LIN {X 0,Y 368.794,Z 449.579,A -85,B 0,C 180,E1 -12880.986,E2 -12880.986} C_VEL
LIN {X 0,Y 368.966,Z 448.589,A -85,B 0,C 180,E1 -12882.095,E2 -12882.095} C_VEL
LIN {X 0,Y 369.505,Z 445.744,A -85,B 0,C 180,E1 -12884.062,E2 -12884.062} C_VEL
LIN {X 0,Y 370.092,Z 441.621,A -85,B 0,C 180,E1 -12885.983,E2 -12885.983} C_VEL
LIN {X 0,Y 370.796,Z 436.818,A -85,B 0,C 180,E1 -12887.654,E2 -12887.654} C_VEL
LIN {X 0,Y 371.622,Z 430.934,A -85,B 0,C 180,E1 -12889.269,E2 -12889.269} C_VEL
LIN {X 0,Y 372.743,Z 423.026,A -85,B 0,C 180,E1 -12890.992,E2 -12890.992} C_VEL
LIN {X 0,Y 373.826,Z 414.283,A -85,B 0,C 180,E1 -12892.509,E2 -12892.509} C_VEL
LIN {X 0,Y 374.877,Z 404.263,A -85,B 0,C 180,E1 -12893.917,E2 -12893.917} C_VEL
LIN {X 0,Y 375.773,Z 395.454,A -85,B 0,C 180,E1 -12894.914,E2 -12894.914} C_VEL
LIN {X 0,Y 375.534,Z 390.642,A -85,B 0,C 180,E1 -12895.44,E2 -12895.44} C_VEL
LIN {X 0,Y 373.509,Z 382.744,A -85,B 0,C 180,E1 -12896.307,E2 -12896.307} C_VEL
LIN {X 0,Y 371.458,Z 374.464,A -85,B 0,C 180,E1 -12897.072,E2 -12897.072} C_VEL
LIN {X 0,Y 371.152,Z 369.066,A -85,B 0,C 180,E1 -12897.429,E2 -12897.429} C_VEL
LIN {X 0,Y 371.504,Z 356.306,A -85,B 0,C 180,E1 -12898.033,E2 -12898.033} C_VEL
LIN {X 0,Y 371.686,Z 343.881,A -85,B 0,C 180,E1 -12898.405,E2 -12898.405} C_VEL
LIN {X 0,Y 372.372,Z 304.643,A -85,B 0,C 180,E1 -12899.179,E2 -12899.179} C_VEL
LIN {X 0,Y 372.772,Z 284.426,A -85,B 0,C 180,E1 -12899.575,E2 -12899.575} C_VEL
LIN {X 0,Y 364.309,Z 266.025,A -85,B 0,C 180,E1 -12900.603,E2 -12900.603} C_VEL
LIN {X 0,Y 362.041,Z 261.256,A -85,B 0,C 180,E1 -12900.916,E2 -12900.916} C_VEL
LIN {X 0,Y 361.882,Z 260.447,A -85,B 0,C 180,E1 -12901.182,E2 -12901.182} C_VEL
LIN {X 0,Y 361.852,Z 260.4,A -85,B 0,C 180,E1 -12904.28,E2 -12904.28} C_VEL
LIN {X 0,Y 361.858,Z 260.37,A -85,B 0,C 180,E1 -12907.221,E2 -12907.221} C_VEL
LIN {X 0,Y 361.811,Z 260.413,A -85,B 0,C 180,E1 -12910.75,E2 -12910.75} C_VEL
LIN {X 0,Y 361.811,Z 260.421,A -85,B 0,C 180,E1 -12914.369,E2 -12914.369} C_VEL
LIN {X 0,Y 361.821,Z 260.402,A -85,B 0,C 180,E1 -12917.57,E2 -12917.57} C_VEL
LIN {X 0,Y 361.84,Z 260.396,A -85,B 0,C 180,E1 -12921.571,E2 -12921.571} C_VEL
LIN {X 0,Y 361.872,Z 260.405,A -85,B 0,C 180,E1 -12924.655,E2 -12924.655} C_VEL
LIN {X 0,Y 361.835,Z 260.392,A -85,B 0,C 180,E1 -12928.37,E2 -12928.37} C_VEL
LIN {X 0,Y 361.863,Z 260.391,A -85,B 0,C 180,E1 -12930.952,E2 -12930.952} C_VEL
LIN {X 0,Y 361.872,Z 260.405,A -85,B 0,C 180,E1 -12934.705,E2 -12934.705} C_VEL
LIN {X 0,Y 361.851,Z 260.373,A -85,B 0,C 180,E1 -12938.344,E2 -12938.344} C_VEL
LIN {X 0,Y 361.964,Z 260.396,A -85,B 0,C 180,E1 -12942.061,E2 -12942.061} C_VEL
LIN {X 0,Y 361.994,Z 260.386,A -85,B 0,C 180,E1 -12946.101,E2 -12946.101} C_VEL
LIN {X 0,Y 361.993,Z 260.384,A -85,B 0,C 180,E1 -12949.937,E2 -12949.937} C_VEL
LIN {X 0,Y 362.112,Z 260.378,A -85,B 0,C 180,E1 -12953.312,E2 -12953.312} C_VEL
LIN {X 0,Y 362.257,Z 260.357,A -85,B 0,C 180,E1 -12957.776,E2 -12957.776} C_VEL
LIN {X 0,Y 362.262,Z 260.35,A -85,B 0,C 180,E1 -12962.223,E2 -12962.223} C_VEL
LIN {X 0,Y 362.109,Z 260.371,A -85,B 0,C 180,E1 -12966.687,E2 -12966.687} C_VEL
LIN {X 0,Y 361.993,Z 260.392,A -85,B 0,C 180,E1 -12970.063,E2 -12970.063} C_VEL
LIN {X 0,Y 361.993,Z 260.387,A -85,B 0,C 180,E1 -12973.899,E2 -12973.899} C_VEL
LIN {X 0,Y 361.922,Z 260.403,A -85,B 0,C 180,E1 -12976.934,E2 -12976.934} C_VEL
LIN {X 0,Y 361.878,Z 260.407,A -85,B 0,C 180,E1 -12980.461,E2 -12980.461} C_VEL
LIN {X 0,Y 361.889,Z 260.406,A -85,B 0,C 180,E1 -12984.113,E2 -12984.113} C_VEL
LIN {X 0,Y 361.83,Z 260.393,A -85,B 0,C 180,E1 -12987.785,E2 -12987.785} C_VEL
LIN {X 0,Y 361.822,Z 260.415,A -85,B 0,C 180,E1 -12991.28,E2 -12991.28} C_VEL
LIN {X 0,Y 361.849,Z 260.396,A -85,B 0,C 180,E1 -12994.281,E2 -12994.281} C_VEL
LIN {X 0,Y 361.854,Z 260.408,A -85,B 0,C 180,E1 -12997.222,E2 -12997.222} C_VEL
LIN {X 0,Y 361.807,Z 260.419,A -85,B 0,C 180,E1 -13000.751,E2 -13000.751} C_VEL
LIN {X 0,Y 361.808,Z 260.415,A -85,B 0,C 180,E1 -13004.37,E2 -13004.37} C_VEL
LIN {X 0,Y 361.819,Z 260.416,A -85,B 0,C 180,E1 -13007.571,E2 -13007.571} C_VEL
LIN {X 0,Y 361.839,Z 260.393,A -85,B 0,C 180,E1 -13011.572,E2 -13011.572} C_VEL
LIN {X 0,Y 361.914,Z 260.609,A -85,B 0,C 180,E1 -13015.283,E2 -13015.283} C_VEL
LIN {X 0,Y 364.922,Z 272.495,A -85,B 0,C 180,E1 -13017.929,E2 -13017.929} C_VEL
LIN {X 0,Y 367.637,Z 284.863,A -85,B 0,C 180,E1 -13020.511,E2 -13020.511} C_VEL
LIN {X 0,Y 367.806,Z 288.203,A -85,B 0,C 180,E1 -13021.153,E2 -13021.153} C_VEL
LIN {X 0,Y 365.998,Z 306.761,A -85,B 0,C 180,E1 -13024.49,E2 -13024.49} C_VEL
LIN {X 0,Y 364.837,Z 320.891,A -85,B 0,C 180,E1 -13026.972,E2 -13026.972} C_VEL
LIN {X 0,Y 369.095,Z 349.309,A -85,B 0,C 180,E1 -13027.909,E2 -13027.909} C_VEL
LIN {X 0,Y 371.223,Z 369.3,A -85,B 0,C 180,E1 -13028.472,E2 -13028.472} C_VEL
LIN {X 0,Y 370.056,Z 432.727,A -85,B 0,C 180,E1 -13029.748,E2 -13029.748} C_VEL
LIN {X 0,Y 369.257,Z 446.633,A -85,B 0,C 180,E1 -13030.255,E2 -13030.255} C_VEL
LIN {X 0,Y 368.138,Z 458.947,A -85,B 0,C 180,E1 -13030.918,E2 -13030.918} C_VEL
LIN {X 0,Y 366.661,Z 471.598,A -85,B 0,C 180,E1 -13031.852,E2 -13031.852} C_VEL
LIN {X 0,Y 365.384,Z 482.905,A -85,B 0,C 180,E1 -13032.943,E2 -13032.943} C_VEL
LIN {X 0,Y 364.037,Z 493.136,A -85,B 0,C 180,E1 -13034.175,E2 -13034.175} C_VEL
LIN {X 0,Y 362.945,Z 503.063,A -85,B 0,C 180,E1 -13035.677,E2 -13035.677} C_VEL
LIN {X 0,Y 361.853,Z 512.169,A -85,B 0,C 180,E1 -13037.379,E2 -13037.379} C_VEL
LIN {X 0,Y 361.162,Z 519.379,A -85,B 0,C 180,E1 -13039.063,E2 -13039.063} C_VEL
LIN {X 0,Y 360.78,Z 526.029,A -85,B 0,C 180,E1 -13041.034,E2 -13041.034} C_VEL
LIN {X 0,Y 360.695,Z 530.466,A -85,B 0,C 180,E1 -13042.724,E2 -13042.724} C_VEL
LIN {X 0,Y 360.828,Z 533.844,A -85,B 0,C 180,E1 -13044.411,E2 -13044.411} C_VEL
LIN {X 0,Y 361.054,Z 536.833,A -85,B 0,C 180,E1 -13046.652,E2 -13046.652} C_VEL
LIN {X 0,Y 361.064,Z 537.659,A -85,B 0,C 180,E1 -13047.769,E2 -13047.769} C_VEL
LIN {X 0,Y 361.187,Z 538.105,A -85,B 0,C 180,E1 -13050,E2 -13050} C_VEL
LIN {X 0,Y 361.135,Z 537.717,A -85,B 0,C 180,E1 -13051.115,E2 -13051.115} C_VEL
LIN {X 0,Y 361.114,Z 536.889,A -85,B 0,C 180,E1 -13052.23,E2 -13052.23} C_VEL
LIN {X 0,Y 361.175,Z 535.642,A -85,B 0,C 180,E1 -13053.346,E2 -13053.346} C_VEL
LIN {X 0,Y 360.962,Z 532.923,A -85,B 0,C 180,E1 -13055.026,E2 -13055.026} C_VEL
LIN {X 0,Y 360.858,Z 529.155,A -85,B 0,C 180,E1 -13056.71,E2 -13056.71} C_VEL
LIN {X 0,Y 360.847,Z 524.233,A -85,B 0,C 180,E1 -13058.399,E2 -13058.399} C_VEL
LIN {X 0,Y 361.024,Z 518.022,A -85,B 0,C 180,E1 -13060.09,E2 -13060.09} C_VEL
LIN {X 0,Y 361.441,Z 510.307,A -85,B 0,C 180,E1 -13061.78,E2 -13061.78} C_VEL
LIN {X 0,Y 362.104,Z 502.46,A -85,B 0,C 180,E1 -13063.182,E2 -13063.182} C_VEL
LIN {X 0,Y 362.746,Z 494.101,A -85,B 0,C 180,E1 -13064.422,E2 -13064.422} C_VEL
LIN {X 0,Y 363.596,Z 483.575,A -85,B 0,C 180,E1 -13065.7,E2 -13065.7} C_VEL
LIN {X 0,Y 364.655,Z 472.11,A -85,B 0,C 180,E1 -13066.803,E2 -13066.803} C_VEL
LIN {X 0,Y 365.687,Z 460.234,A -85,B 0,C 180,E1 -13067.691,E2 -13067.691} C_VEL
LIN {X 0,Y 366.606,Z 447.205,A -85,B 0,C 180,E1 -13068.403,E2 -13068.403} C_VEL
LIN {X 0,Y 367.2,Z 433.206,A -85,B 0,C 180,E1 -13068.915,E2 -13068.915} C_VEL
LIN {X 0,Y 368.032,Z 367.575,A -85,B 0,C 180,E1 -13070.214,E2 -13070.214} C_VEL
LIN {X 0,Y 363.351,Z 322.227,A -85,B 0,C 180,E1 -13071.372,E2 -13071.372} C_VEL
LIN {X 0,Y 365.027,Z 297.412,A -85,B 0,C 180,E1 -13075.669,E2 -13075.669} C_VEL
LIN {X 0,Y 366.152,Z 281.581,A -85,B 0,C 180,E1 -13078.452,E2 -13078.452} C_VEL
LIN {X 0,Y 363.857,Z 269.465,A -85,B 0,C 180,E1 -13080.786,E2 -13080.786} C_VEL
LIN {X 0,Y 361.881,Z 260.54,A -85,B 0,C 180,E1 -13082.609,E2 -13082.609} C_VEL
LIN {X 0,Y 361.858,Z 260.411,A -85,B 0,C 180,E1 -13085.636,E2 -13085.636} C_VEL
LIN {X 0,Y 361.818,Z 260.415,A -85,B 0,C 180,E1 -13089.016,E2 -13089.016} C_VEL
LIN {X 0,Y 361.822,Z 260.413,A -85,B 0,C 180,E1 -13092.829,E2 -13092.829} C_VEL
LIN {X 0,Y 361.805,Z 260.414,A -85,B 0,C 180,E1 -13095.947,E2 -13095.947} C_VEL
LIN {X 0,Y 361.802,Z 260.419,A -85,B 0,C 180,E1 -13099.248,E2 -13099.248} C_VEL
LIN {X 0,Y 361.852,Z 260.412,A -85,B 0,C 180,E1 -13102.98,E2 -13102.98} C_VEL
LIN {X 0,Y 361.848,Z 260.41,A -85,B 0,C 180,E1 -13106.631,E2 -13106.631} C_VEL
LIN {X 0,Y 361.837,Z 260.41,A -85,B 0,C 180,E1 -13109.669,E2 -13109.669} C_VEL
LIN {X 0,Y 361.843,Z 260.41,A -85,B 0,C 180,E1 -13113.466,E2 -13113.466} C_VEL
LIN {X 0,Y 361.859,Z 260.407,A -85,B 0,C 180,E1 -13115.93,E2 -13115.93} C_VEL
LIN {X 0,Y 361.865,Z 260.407,A -85,B 0,C 180,E1 -13119.538,E2 -13119.538} C_VEL
LIN {X 0,Y 361.915,Z 260.403,A -85,B 0,C 180,E1 -13123.065,E2 -13123.065} C_VEL
LIN {X 0,Y 361.988,Z 260.395,A -85,B 0,C 180,E1 -13126.528,E2 -13126.528} C_VEL
LIN {X 0,Y 361.985,Z 260.391,A -85,B 0,C 180,E1 -13129.937,E2 -13129.937} C_VEL
LIN {X 0,Y 362.103,Z 260.377,A -85,B 0,C 180,E1 -13133.313,E2 -13133.313} C_VEL
LIN {X 0,Y 362.255,Z 260.358,A -85,B 0,C 180,E1 -13137.777,E2 -13137.777} C_VEL
LIN {X 0,Y 362.244,Z 260.362,A -85,B 0,C 180,E1 -13142.224,E2 -13142.224} C_VEL
LIN {X 0,Y 362.106,Z 260.379,A -85,B 0,C 180,E1 -13146.688,E2 -13146.688} C_VEL
LIN {X 0,Y 361.982,Z 260.395,A -85,B 0,C 180,E1 -13150.064,E2 -13150.064} C_VEL
LIN {X 0,Y 361.988,Z 260.393,A -85,B 0,C 180,E1 -13153.899,E2 -13153.899} C_VEL
LIN {X 0,Y 361.917,Z 260.4,A -85,B 0,C 180,E1 -13156.935,E2 -13156.935} C_VEL
LIN {X 0,Y 361.874,Z 260.408,A -85,B 0,C 180,E1 -13160.462,E2 -13160.462} C_VEL
LIN {X 0,Y 361.852,Z 260.414,A -85,B 0,C 180,E1 -13164.102,E2 -13164.102} C_VEL
LIN {X 0,Y 361.826,Z 260.414,A -85,B 0,C 180,E1 -13167.786,E2 -13167.786} C_VEL
LIN {X 0,Y 361.839,Z 260.41,A -85,B 0,C 180,E1 -13171.286,E2 -13171.286} C_VEL
LIN {X 0,Y 361.843,Z 260.412,A -85,B 0,C 180,E1 -13174.282,E2 -13174.282} C_VEL
LIN {X 0,Y 361.85,Z 260.409,A -85,B 0,C 180,E1 -13177.222,E2 -13177.222} C_VEL
LIN {X 0,Y 361.804,Z 260.414,A -85,B 0,C 180,E1 -13180.752,E2 -13180.752} C_VEL
LIN {X 0,Y 361.805,Z 260.414,A -85,B 0,C 180,E1 -13184.371,E2 -13184.371} C_VEL
LIN {X 0,Y 361.817,Z 260.417,A -85,B 0,C 180,E1 -13187.572,E2 -13187.572} C_VEL
LIN {X 0,Y 361.838,Z 260.415,A -85,B 0,C 180,E1 -13191.573,E2 -13191.573} C_VEL
LIN {X 0,Y 361.867,Z 260.406,A -85,B 0,C 180,E1 -13194.658,E2 -13194.658} C_VEL
LIN {X 0,Y 361.844,Z 260.41,A -85,B 0,C 180,E1 -13197.056,E2 -13197.056} C_VEL
LIN {X 0,Y 361.848,Z 260.409,A -85,B 0,C 180,E1 -13200.952,E2 -13200.952} C_VEL
LIN {X 0,Y 361.859,Z 260.407,A -85,B 0,C 180,E1 -13204.706,E2 -13204.706} C_VEL
LIN {X 0,Y 361.86,Z 260.407,A -85,B 0,C 180,E1 -13208.346,E2 -13208.346} C_VEL
LIN {X 0,Y 361.906,Z 260.401,A -85,B 0,C 180,E1 -13212.094,E2 -13212.094} C_VEL
LIN {X 0,Y 361.953,Z 260.389,A -85,B 0,C 180,E1 -13216.133,E2 -13216.133} C_VEL
LIN {X 0,Y 362.035,Z 260.634,A -85,B 0,C 180,E1 -13216.958,E2 -13216.958} C_VEL
LIN {X 0,Y 362.301,Z 261.741,A -85,B 0,C 180,E1 -13217.125,E2 -13217.125} C_VEL
LIN {X 0,Y 369.26,Z 280.308,A -85,B 0,C 180,E1 -13217.878,E2 -13217.878} C_VEL
LIN {X 0,Y 368.244,Z 347.877,A -85,B 0,C 180,E1 -13219.207,E2 -13219.207} C_VEL
LIN {X 0,Y 368.066,Z 360.994,A -85,B 0,C 180,E1 -13219.689,E2 -13219.689} C_VEL
LIN {X 0,Y 367.703,Z 372.477,A -85,B 0,C 180,E1 -13220.304,E2 -13220.304} C_VEL
LIN {X 0,Y 367.062,Z 384.829,A -85,B 0,C 180,E1 -13221.19,E2 -13221.19} C_VEL
LIN {X 0,Y 366.27,Z 396.386,A -85,B 0,C 180,E1 -13222.282,E2 -13222.282} C_VEL
LIN {X 0,Y 365.484,Z 406.742,A -85,B 0,C 180,E1 -13223.514,E2 -13223.514} C_VEL
LIN {X 0,Y 364.793,Z 415.21,A -85,B 0,C 180,E1 -13224.75,E2 -13224.75} C_VEL
LIN {X 0,Y 364.094,Z 423.021,A -85,B 0,C 180,E1 -13226.127,E2 -13226.127} C_VEL
LIN {X 0,Y 363.274,Z 430.704,A -85,B 0,C 180,E1 -13227.783,E2 -13227.783} C_VEL
LIN {X 0,Y 362.656,Z 436.84,A -85,B 0,C 180,E1 -13229.445,E2 -13229.445} C_VEL
LIN {X 0,Y 362.193,Z 441.726,A -85,B 0,C 180,E1 -13231.112,E2 -13231.112} C_VEL
LIN {X 0,Y 361.837,Z 445.517,A -85,B 0,C 180,E1 -13232.784,E2 -13232.784} C_VEL
LIN {X 0,Y 361.658,Z 448.299,A -85,B 0,C 180,E1 -13234.459,E2 -13234.459} C_VEL
LIN {X 0,Y 361.626,Z 449.614,A -85,B 0,C 180,E1 -13235.577,E2 -13235.577} C_VEL
LIN {X 0,Y 361.569,Z 451.113,A -85,B 0,C 180,E1 -13237.82,E2 -13237.82} C_VEL
LIN {X 0,Y 361.68,Z 450.991,A -85,B 0,C 180,E1 -13240.072,E2 -13240.072} C_VEL
LIN {X 0,Y 361.797,Z 450.359,A -85,B 0,C 180,E1 -13241.201,E2 -13241.201} C_VEL
LIN {X 0,Y 361.982,Z 449.329,A -85,B 0,C 180,E1 -13242.332,E2 -13242.332} C_VEL
LIN {X 0,Y 362.531,Z 446.595,A -85,B 0,C 180,E1 -13244.232,E2 -13244.232} C_VEL
LIN {X 0,Y 363.212,Z 442.213,A -85,B 0,C 180,E1 -13246.294,E2 -13246.294} C_VEL
LIN {X 0,Y 363.955,Z 437.339,A -85,B 0,C 180,E1 -13247.997,E2 -13247.997} C_VEL
LIN {X 0,Y 364.868,Z 431.376,A -85,B 0,C 180,E1 -13249.641,E2 -13249.641} C_VEL
LIN {X 0,Y 365.853,Z 424.772,A -85,B 0,C 180,E1 -13251.112,E2 -13251.112} C_VEL
LIN {X 0,Y 367.027,Z 415.918,A -85,B 0,C 180,E1 -13252.709,E2 -13252.709} C_VEL
LIN {X 0,Y 368.04,Z 406.472,A -85,B 0,C 180,E1 -13254.09,E2 -13254.09} C_VEL
LIN {X 0,Y 369.221,Z 395.597,A -85,B 0,C 180,E1 -13255.358,E2 -13255.358} C_VEL
LIN {X 0,Y 370.101,Z 385.806,A -85,B 0,C 180,E1 -13256.27,E2 -13256.27} C_VEL
LIN {X 0,Y 370.899,Z 374.104,A -85,B 0,C 180,E1 -13257.126,E2 -13257.126} C_VEL
LIN {X 0,Y 371.152,Z 369.066,A -85,B 0,C 180,E1 -13257.429,E2 -13257.429} C_VEL
LIN {X 0,Y 370.716,Z 365.396,A -85,B 0,C 180,E1 -13257.67,E2 -13257.67} C_VEL
LIN {X 0,Y 365.698,Z 354.113,A -85,B 0,C 180,E1 -13258.532,E2 -13258.532} C_VEL
LIN {X 0,Y 365.154,Z 350.323,A -85,B 0,C 180,E1 -13258.697,E2 -13258.697} C_VEL
LIN {X 0,Y 365.736,Z 311.849,A -85,B 0,C 180,E1 -13259.507,E2 -13259.507} C_VEL
LIN {X 0,Y 366.277,Z 286.132,A -85,B 0,C 180,E1 -13260.019,E2 -13260.019} C_VEL
LIN {X 0,Y 357.814,Z 267.909,A -85,B 0,C 180,E1 -13261.076,E2 -13261.076} C_VEL
LIN {X 0,Y 355.007,Z 262.187,A -85,B 0,C 180,E1 -13261.458,E2 -13261.458} C_VEL
LIN {X 0,Y 354.799,Z 261.368,A -85,B 0,C 180,E1 -13261.702,E2 -13261.702} C_VEL
LIN {X 0,Y 354.809,Z 261.256,A -85,B 0,C 180,E1 -13265.059,E2 -13265.059} C_VEL
LIN {X 0,Y 354.793,Z 261.258,A -85,B 0,C 180,E1 -13267.884,E2 -13267.884} C_VEL
LIN {X 0,Y 354.769,Z 261.286,A -85,B 0,C 180,E1 -13271.167,E2 -13271.167} C_VEL
LIN {X 0,Y 354.758,Z 261.299,A -85,B 0,C 180,E1 -13274.505,E2 -13274.505} C_VEL
LIN {X 0,Y 354.78,Z 261.279,A -85,B 0,C 180,E1 -13277.66,E2 -13277.66} C_VEL
LIN {X 0,Y 354.784,Z 261.284,A -85,B 0,C 180,E1 -13280.661,E2 -13280.661} C_VEL
LIN {X 0,Y 354.819,Z 261.278,A -85,B 0,C 180,E1 -13284.3,E2 -13284.3} C_VEL
LIN {X 0,Y 354.785,Z 261.281,A -85,B 0,C 180,E1 -13287.666,E2 -13287.666} C_VEL
LIN {X 0,Y 354.796,Z 261.279,A -85,B 0,C 180,E1 -13291.614,E2 -13291.614} C_VEL
LIN {X 0,Y 354.837,Z 261.279,A -85,B 0,C 180,E1 -13295.422,E2 -13295.422} C_VEL
LIN {X 0,Y 354.821,Z 261.253,A -85,B 0,C 180,E1 -13299.112,E2 -13299.112} C_VEL
LIN {X 0,Y 354.895,Z 261.277,A -85,B 0,C 180,E1 -13302.719,E2 -13302.719} C_VEL
LIN {X 0,Y 354.947,Z 261.265,A -85,B 0,C 180,E1 -13306.255,E2 -13306.255} C_VEL
LIN {X 0,Y 354.95,Z 261.263,A -85,B 0,C 180,E1 -13309.735,E2 -13309.735} C_VEL
LIN {X 0,Y 355.079,Z 261.253,A -85,B 0,C 180,E1 -13313.179,E2 -13313.179} C_VEL
LIN {X 0,Y 355.219,Z 261.233,A -85,B 0,C 180,E1 -13317.732,E2 -13317.732} C_VEL
LIN {X 0,Y 355.139,Z 261.239,A -85,B 0,C 180,E1 -13321.134,E2 -13321.134} C_VEL
LIN {X 0,Y 355.224,Z 261.226,A -85,B 0,C 180,E1 -13322.268,E2 -13322.268} C_VEL
LIN {X 0,Y 355.076,Z 261.247,A -85,B 0,C 180,E1 -13326.82,E2 -13326.82} C_VEL
LIN {X 0,Y 354.949,Z 261.269,A -85,B 0,C 180,E1 -13330.265,E2 -13330.265} C_VEL
LIN {X 0,Y 354.938,Z 261.267,A -85,B 0,C 180,E1 -13334.018,E2 -13334.018} C_VEL
LIN {X 0,Y 354.885,Z 261.272,A -85,B 0,C 180,E1 -13338.092,E2 -13338.092} C_VEL
LIN {X 0,Y 354.812,Z 261.284,A -85,B 0,C 180,E1 -13341.417,E2 -13341.417} C_VEL
LIN {X 0,Y 354.843,Z 261.284,A -85,B 0,C 180,E1 -13344.577,E2 -13344.577} C_VEL
LIN {X 0,Y 354.784,Z 261.274,A -85,B 0,C 180,E1 -13348.387,E2 -13348.387} C_VEL
LIN {X 0,Y 354.775,Z 261.288,A -85,B 0,C 180,E1 -13352.335,E2 -13352.335} C_VEL
LIN {X 0,Y 354.817,Z 261.287,A -85,B 0,C 180,E1 -13355.699,E2 -13355.699} C_VEL
LIN {X 0,Y 354.765,Z 261.285,A -85,B 0,C 180,E1 -13359.413,E2 -13359.413} C_VEL
LIN {X 0,Y 354.778,Z 261.285,A -85,B 0,C 180,E1 -13362.866,E2 -13362.866} C_VEL
LIN {X 0,Y 354.759,Z 261.29,A -85,B 0,C 180,E1 -13366.103,E2 -13366.103} C_VEL
LIN {X 0,Y 354.76,Z 261.286,A -85,B 0,C 180,E1 -13369.176,E2 -13369.176} C_VEL
LIN {X 0,Y 354.796,Z 261.284,A -85,B 0,C 180,E1 -13372.405,E2 -13372.405} C_VEL
LIN {X 0,Y 354.867,Z 261.516,A -85,B 0,C 180,E1 -13374.808,E2 -13374.808} C_VEL
LIN {X 0,Y 357.964,Z 273.72,A -85,B 0,C 180,E1 -13377.59,E2 -13377.59} C_VEL
LIN {X 0,Y 360.672,Z 285.936,A -85,B 0,C 180,E1 -13380.206,E2 -13380.206} C_VEL
LIN {X 0,Y 361.002,Z 289.292,A -85,B 0,C 180,E1 -13380.876,E2 -13380.876} C_VEL
LIN {X 0,Y 359.358,Z 305.33,A -85,B 0,C 180,E1 -13383.817,E2 -13383.817} C_VEL
LIN {X 0,Y 358.071,Z 319.999,A -85,B 0,C 180,E1 -13386.444,E2 -13386.444} C_VEL
LIN {X 0,Y 362.388,Z 348.333,A -85,B 0,C 180,E1 -13387.415,E2 -13387.415} C_VEL
LIN {X 0,Y 364.682,Z 369.563,A -85,B 0,C 180,E1 -13388.031,E2 -13388.031} C_VEL
LIN {X 0,Y 363.49,Z 431.442,A -85,B 0,C 180,E1 -13389.293,E2 -13389.293} C_VEL
LIN {X 0,Y 362.782,Z 444.691,A -85,B 0,C 180,E1 -13389.777,E2 -13389.777} C_VEL
LIN {X 0,Y 361.649,Z 456.751,A -85,B 0,C 180,E1 -13390.414,E2 -13390.414} C_VEL
LIN {X 0,Y 360.359,Z 468.169,A -85,B 0,C 180,E1 -13391.228,E2 -13391.228} C_VEL
LIN {X 0,Y 358.911,Z 479.95,A -85,B 0,C 180,E1 -13392.331,E2 -13392.331} C_VEL
LIN {X 0,Y 357.475,Z 490.561,A -85,B 0,C 180,E1 -13393.584,E2 -13393.584} C_VEL
LIN {X 0,Y 356.349,Z 499.279,A -85,B 0,C 180,E1 -13394.852,E2 -13394.852} C_VEL
LIN {X 0,Y 355.493,Z 507.367,A -85,B 0,C 180,E1 -13396.276,E2 -13396.276} C_VEL
LIN {X 0,Y 354.644,Z 514.098,A -85,B 0,C 180,E1 -13397.7,E2 -13397.7} C_VEL
LIN {X 0,Y 353.935,Z 520.776,A -85,B 0,C 180,E1 -13399.416,E2 -13399.416} C_VEL
LIN {X 0,Y 353.667,Z 526.917,A -85,B 0,C 180,E1 -13401.429,E2 -13401.429} C_VEL
LIN {X 0,Y 353.709,Z 531.549,A -85,B 0,C 180,E1 -13403.451,E2 -13403.451} C_VEL
LIN {X 0,Y 353.808,Z 534.75,A -85,B 0,C 180,E1 -13405.442,E2 -13405.442} C_VEL
LIN {X 0,Y 353.977,Z 536.023,A -85,B 0,C 180,E1 -13406.585,E2 -13406.585} C_VEL
LIN {X 0,Y 354.014,Z 536.829,A -85,B 0,C 180,E1 -13407.724,E2 -13407.724} C_VEL
LIN {X 0,Y 354.138,Z 537.248,A -85,B 0,C 180,E1 -13410,E2 -13410} C_VEL
LIN {X 0,Y 354.084,Z 536.842,A -85,B 0,C 180,E1 -13411.137,E2 -13411.137} C_VEL
LIN {X 0,Y 354.064,Z 535.988,A -85,B 0,C 180,E1 -13412.275,E2 -13412.275} C_VEL
LIN {X 0,Y 354.129,Z 534.725,A -85,B 0,C 180,E1 -13413.413,E2 -13413.413} C_VEL
LIN {X 0,Y 353.882,Z 531.968,A -85,B 0,C 180,E1 -13415.127,E2 -13415.127} C_VEL
LIN {X 0,Y 353.771,Z 528.163,A -85,B 0,C 180,E1 -13416.845,E2 -13416.845} C_VEL
LIN {X 0,Y 353.776,Z 523.202,A -85,B 0,C 180,E1 -13418.568,E2 -13418.568} C_VEL
LIN {X 0,Y 353.963,Z 516.946,A -85,B 0,C 180,E1 -13420.293,E2 -13420.293} C_VEL
LIN {X 0,Y 354.412,Z 509.183,A -85,B 0,C 180,E1 -13422.017,E2 -13422.017} C_VEL
LIN {X 0,Y 355.112,Z 501.278,A -85,B 0,C 180,E1 -13423.446,E2 -13423.446} C_VEL
LIN {X 0,Y 355.76,Z 493.258,A -85,B 0,C 180,E1 -13424.654,E2 -13424.654} C_VEL
LIN {X 0,Y 356.593,Z 483.526,A -85,B 0,C 180,E1 -13425.869,E2 -13425.869} C_VEL
LIN {X 0,Y 357.66,Z 472.237,A -85,B 0,C 180,E1 -13426.994,E2 -13426.994} C_VEL
LIN {X 0,Y 358.829,Z 459.612,A -85,B 0,C 180,E1 -13427.967,E2 -13427.967} C_VEL
LIN {X 0,Y 359.731,Z 446.686,A -85,B 0,C 180,E1 -13428.694,E2 -13428.694} C_VEL
LIN {X 0,Y 360.329,Z 434.005,A -85,B 0,C 180,E1 -13429.178,E2 -13429.178} C_VEL
LIN {X 0,Y 360.743,Z 410.493,A -85,B 0,C 180,E1 -13429.688,E2 -13429.688} C_VEL
LIN {X 0,Y 361.236,Z 368.258,A -85,B 0,C 180,E1 -13430.523,E2 -13430.523} C_VEL
LIN {X 0,Y 356.406,Z 321.507,A -85,B 0,C 180,E1 -13431.736,E2 -13431.736} C_VEL
LIN {X 0,Y 357.944,Z 299.576,A -85,B 0,C 180,E1 -13435.591,E2 -13435.591} C_VEL
LIN {X 0,Y 359.183,Z 283.797,A -85,B 0,C 180,E1 -13438.413,E2 -13438.413} C_VEL
LIN {X 0,Y 358.559,Z 278.956,A -85,B 0,C 180,E1 -13439.34,E2 -13439.34} C_VEL
LIN {X 0,Y 355.509,Z 264.371,A -85,B 0,C 180,E1 -13442.258,E2 -13442.258} C_VEL
LIN {X 0,Y 354.823,Z 261.415,A -85,B 0,C 180,E1 -13442.918,E2 -13442.918} C_VEL
LIN {X 0,Y 354.786,Z 261.288,A -85,B 0,C 180,E1 -13446.459,E2 -13446.459} C_VEL
LIN {X 0,Y 354.763,Z 261.296,A -85,B 0,C 180,E1 -13449.411,E2 -13449.411} C_VEL
LIN {X 0,Y 354.774,Z 261.292,A -85,B 0,C 180,E1 -13452.865,E2 -13452.865} C_VEL
LIN {X 0,Y 354.754,Z 261.291,A -85,B 0,C 180,E1 -13456.102,E2 -13456.102} C_VEL
LIN {X 0,Y 354.755,Z 261.298,A -85,B 0,C 180,E1 -13459.175,E2 -13459.175} C_VEL
LIN {X 0,Y 354.79,Z 261.287,A -85,B 0,C 180,E1 -13462.404,E2 -13462.404} C_VEL
LIN {X 0,Y 354.799,Z 261.291,A -85,B 0,C 180,E1 -13464.939,E2 -13464.939} C_VEL
LIN {X 0,Y 354.766,Z 261.29,A -85,B 0,C 180,E1 -13468.409,E2 -13468.409} C_VEL
LIN {X 0,Y 354.778,Z 261.29,A -85,B 0,C 180,E1 -13471.613,E2 -13471.613} C_VEL
LIN {X 0,Y 354.824,Z 261.283,A -85,B 0,C 180,E1 -13475.657,E2 -13475.657} C_VEL
LIN {X 0,Y 354.811,Z 261.288,A -85,B 0,C 180,E1 -13479.112,E2 -13479.112} C_VEL
LIN {X 0,Y 354.868,Z 261.282,A -85,B 0,C 180,E1 -13482.719,E2 -13482.719} C_VEL
LIN {X 0,Y 354.94,Z 261.27,A -85,B 0,C 180,E1 -13486.255,E2 -13486.255} C_VEL
LIN {X 0,Y 354.941,Z 261.268,A -85,B 0,C 180,E1 -13489.735,E2 -13489.735} C_VEL
LIN {X 0,Y 355.07,Z 261.254,A -85,B 0,C 180,E1 -13493.18,E2 -13493.18} C_VEL
LIN {X 0,Y 355.217,Z 261.234,A -85,B 0,C 180,E1 -13497.732,E2 -13497.732} C_VEL
LIN {X 0,Y 355.158,Z 261.242,A -85,B 0,C 180,E1 -13501.134,E2 -13501.134} C_VEL
LIN {X 0,Y 355.206,Z 261.239,A -85,B 0,C 180,E1 -13502.268,E2 -13502.268} C_VEL
LIN {X 0,Y 355.072,Z 261.254,A -85,B 0,C 180,E1 -13506.821,E2 -13506.821} C_VEL
LIN {X 0,Y 354.939,Z 261.274,A -85,B 0,C 180,E1 -13510.266,E2 -13510.266} C_VEL
LIN {X 0,Y 354.932,Z 261.273,A -85,B 0,C 180,E1 -13514.019,E2 -13514.019} C_VEL
LIN {X 0,Y 354.881,Z 261.28,A -85,B 0,C 180,E1 -13518.093,E2 -13518.093} C_VEL
LIN {X 0,Y 354.804,Z 261.292,A -85,B 0,C 180,E1 -13522.108,E2 -13522.108} C_VEL
LIN {X 0,Y 354.793,Z 261.29,A -85,B 0,C 180,E1 -13525.836,E2 -13525.836} C_VEL
LIN {X 0,Y 354.785,Z 261.291,A -85,B 0,C 180,E1 -13529.685,E2 -13529.685} C_VEL
LIN {X 0,Y 354.779,Z 261.291,A -85,B 0,C 180,E1 -13532.335,E2 -13532.335} C_VEL
LIN {X 0,Y 354.811,Z 261.288,A -85,B 0,C 180,E1 -13535.699,E2 -13535.699} C_VEL
LIN {X 0,Y 354.762,Z 261.293,A -85,B 0,C 180,E1 -13539.414,E2 -13539.414} C_VEL
LIN {X 0,Y 354.775,Z 261.287,A -85,B 0,C 180,E1 -13542.867,E2 -13542.867} C_VEL
LIN {X 0,Y 354.757,Z 261.294,A -85,B 0,C 180,E1 -13546.104,E2 -13546.104} C_VEL
LIN {X 0,Y 354.758,Z 261.293,A -85,B 0,C 180,E1 -13549.177,E2 -13549.177} C_VEL
LIN {X 0,Y 354.795,Z 261.285,A -85,B 0,C 180,E1 -13552.406,E2 -13552.406} C_VEL
LIN {X 0,Y 354.805,Z 261.286,A -85,B 0,C 180,E1 -13554.942,E2 -13554.942} C_VEL
LIN {X 0,Y 354.774,Z 261.289,A -85,B 0,C 180,E1 -13558.411,E2 -13558.411} C_VEL
LIN {X 0,Y 354.787,Z 261.293,A -85,B 0,C 180,E1 -13561.615,E2 -13561.615} C_VEL
LIN {X 0,Y 354.804,Z 261.291,A -85,B 0,C 180,E1 -13565.421,E2 -13565.421} C_VEL
LIN {X 0,Y 354.82,Z 261.287,A -85,B 0,C 180,E1 -13569.114,E2 -13569.114} C_VEL
LIN {X 0,Y 354.852,Z 261.281,A -85,B 0,C 180,E1 -13572.718,E2 -13572.718} C_VEL
LIN {X 0,Y 354.967,Z 261.43,A -85,B 0,C 180,E1 -13576.548,E2 -13576.548} C_VEL
LIN {X 0,Y 355.229,Z 262.533,A -85,B 0,C 180,E1 -13576.748,E2 -13576.748} C_VEL
LIN {X 0,Y 362.316,Z 281.131,A -85,B 0,C 180,E1 -13577.535,E2 -13577.535} C_VEL
LIN {X 0,Y 361.46,Z 348.669,A -85,B 0,C 180,E1 -13578.896,E2 -13578.896} C_VEL
LIN {X 0,Y 361.28,Z 361.801,A -85,B 0,C 180,E1 -13579.386,E2 -13579.386} C_VEL
LIN {X 0,Y 360.919,Z 372.74,A -85,B 0,C 180,E1 -13579.978,E2 -13579.978} C_VEL
LIN {X 0,Y 360.269,Z 385.221,A -85,B 0,C 180,E1 -13580.881,E2 -13580.881} C_VEL
LIN {X 0,Y 359.439,Z 396.896,A -85,B 0,C 180,E1 -13581.993,E2 -13581.993} C_VEL
LIN {X 0,Y 358.611,Z 407.313,A -85,B 0,C 180,E1 -13583.248,E2 -13583.248} C_VEL
LIN {X 0,Y 357.825,Z 416.699,A -85,B 0,C 180,E1 -13584.647,E2 -13584.647} C_VEL
LIN {X 0,Y 357.096,Z 424.404,A -85,B 0,C 180,E1 -13586.051,E2 -13586.051} C_VEL
LIN {X 0,Y 356.249,Z 431.955,A -85,B 0,C 180,E1 -13587.739,E2 -13587.739} C_VEL
LIN {X 0,Y 355.625,Z 438.014,A -85,B 0,C 180,E1 -13589.434,E2 -13589.434} C_VEL
LIN {X 0,Y 355.154,Z 442.831,A -85,B 0,C 180,E1 -13591.134,E2 -13591.134} C_VEL
LIN {X 0,Y 354.791,Z 446.558,A -85,B 0,C 180,E1 -13592.839,E2 -13592.839} C_VEL
LIN {X 0,Y 354.616,Z 449.279,A -85,B 0,C 180,E1 -13594.547,E2 -13594.547} C_VEL
LIN {X 0,Y 354.576,Z 450.567,A -85,B 0,C 180,E1 -13595.688,E2 -13595.688} C_VEL
LIN {X 0,Y 354.537,Z 451.859,A -85,B 0,C 180,E1 -13597.623,E2 -13597.623} C_VEL
LIN {X 0,Y 354.565,Z 452.083,A -85,B 0,C 180,E1 -13599.124,E2 -13599.124} C_VEL
LIN {X 0,Y 354.811,Z 451.139,A -85,B 0,C 180,E1 -13601.425,E2 -13601.425} C_VEL
LIN {X 0,Y 355.003,Z 450.053,A -85,B 0,C 180,E1 -13602.578,E2 -13602.578} C_VEL
LIN {X 0,Y 355.572,Z 447.433,A -85,B 0,C 180,E1 -13604.416,E2 -13604.416} C_VEL
LIN {X 0,Y 356.331,Z 442.808,A -85,B 0,C 180,E1 -13606.618,E2 -13606.618} C_VEL
LIN {X 0,Y 357.131,Z 437.863,A -85,B 0,C 180,E1 -13608.353,E2 -13608.353} C_VEL
LIN {X 0,Y 358.156,Z 431.579,A -85,B 0,C 180,E1 -13610.084,E2 -13610.084} C_VEL
LIN {X 0,Y 359.347,Z 423.639,A -85,B 0,C 180,E1 -13611.814,E2 -13611.814} C_VEL
LIN {X 0,Y 360.484,Z 415.52,A -85,B 0,C 180,E1 -13613.247,E2 -13613.247} C_VEL
LIN {X 0,Y 361.619,Z 405.455,A -85,B 0,C 180,E1 -13614.699,E2 -13614.699} C_VEL
LIN {X 0,Y 362.696,Z 395.415,A -85,B 0,C 180,E1 -13615.848,E2 -13615.848} C_VEL
LIN {X 0,Y 363.713,Z 384.542,A -85,B 0,C 180,E1 -13616.839,E2 -13616.839} C_VEL
LIN {X 0,Y 364.415,Z 374.426,A -85,B 0,C 180,E1 -13617.571,E2 -13617.571} C_VEL
LIN {X 0,Y 364.932,Z 361.686,A -85,B 0,C 180,E1 -13618.27,E2 -13618.27} C_VEL
LIN {X 0,Y 365.154,Z 350.323,A -85,B 0,C 180,E1 -13618.697,E2 -13618.697} C_VEL
LIN {X 0,Y 364.696,Z 344.57,A -85,B 0,C 180,E1 -13618.899,E2 -13618.899} C_VEL
LIN {X 0,Y 359.585,Z 326.01,A -85,B 0,C 180,E1 -13619.668,E2 -13619.668} C_VEL
LIN {X 0,Y 359.093,Z 320.207,A -85,B 0,C 180,E1 -13619.824,E2 -13619.824} C_VEL
LIN {X 0,Y 359.844,Z 288.07,A -85,B 0,C 180,E1 -13620.47,E2 -13620.47} C_VEL
LIN {X 0,Y 351.908,Z 271.09,A -85,B 0,C 180,E1 -13621.49,E2 -13621.49} C_VEL
LIN {X 0,Y 347.975,Z 263.262,A -85,B 0,C 180,E1 -13622.02,E2 -13622.02} C_VEL
LIN {X 0,Y 347.789,Z 262.295,A -85,B 0,C 180,E1 -13622.239,E2 -13622.239} C_VEL
LIN {X 0,Y 347.767,Z 262.12,A -85,B 0,C 180,E1 -13626.063,E2 -13626.063} C_VEL
LIN {X 0,Y 347.731,Z 262.158,A -85,B 0,C 180,E1 -13628.795,E2 -13628.795} C_VEL
LIN {X 0,Y 347.742,Z 262.156,A -85,B 0,C 180,E1 -13631.831,E2 -13631.831} C_VEL
LIN {X 0,Y 347.7,Z 262.173,A -85,B 0,C 180,E1 -13635.027,E2 -13635.027} C_VEL
LIN {X 0,Y 347.737,Z 262.163,A -85,B 0,C 180,E1 -13638.399,E2 -13638.399} C_VEL
LIN {X 0,Y 347.76,Z 262.144,A -85,B 0,C 180,E1 -13642.013,E2 -13642.013} C_VEL
LIN {X 0,Y 347.743,Z 262.169,A -85,B 0,C 180,E1 -13645.535,E2 -13645.535} C_VEL
LIN {X 0,Y 347.742,Z 262.147,A -85,B 0,C 180,E1 -13648.3,E2 -13648.3} C_VEL
LIN {X 0,Y 347.742,Z 262.148,A -85,B 0,C 180,E1 -13650.984,E2 -13650.984} C_VEL
LIN {X 0,Y 347.743,Z 262.17,A -85,B 0,C 180,E1 -13653.6,E2 -13653.6} C_VEL
LIN {X 0,Y 347.753,Z 262.147,A -85,B 0,C 180,E1 -13656.159,E2 -13656.159} C_VEL
LIN {X 0,Y 347.801,Z 262.136,A -85,B 0,C 180,E1 -13659.908,E2 -13659.908} C_VEL
LIN {X 0,Y 347.863,Z 262.155,A -85,B 0,C 180,E1 -13662.359,E2 -13662.359} C_VEL
LIN {X 0,Y 347.894,Z 262.141,A -85,B 0,C 180,E1 -13665.97,E2 -13665.97} C_VEL
LIN {X 0,Y 347.89,Z 262.145,A -85,B 0,C 180,E1 -13669.524,E2 -13669.524} C_VEL
LIN {X 0,Y 348.046,Z 262.128,A -85,B 0,C 180,E1 -13673.041,E2 -13673.041} C_VEL
LIN {X 0,Y 348.18,Z 262.109,A -85,B 0,C 180,E1 -13677.686,E2 -13677.686} C_VEL
LIN {X 0,Y 348.11,Z 262.114,A -85,B 0,C 180,E1 -13681.157,E2 -13681.157} C_VEL
LIN {X 0,Y 348.186,Z 262.103,A -85,B 0,C 180,E1 -13682.313,E2 -13682.313} C_VEL
LIN {X 0,Y 348.043,Z 262.121,A -85,B 0,C 180,E1 -13686.959,E2 -13686.959} C_VEL
LIN {X 0,Y 347.889,Z 262.148,A -85,B 0,C 180,E1 -13690.475,E2 -13690.475} C_VEL
LIN {X 0,Y 347.894,Z 262.145,A -85,B 0,C 180,E1 -13694.15,E2 -13694.15} C_VEL
LIN {X 0,Y 347.825,Z 262.151,A -85,B 0,C 180,E1 -13698.259,E2 -13698.259} C_VEL
LIN {X 0,Y 347.758,Z 262.161,A -85,B 0,C 180,E1 -13701.624,E2 -13701.624} C_VEL
LIN {X 0,Y 347.761,Z 262.164,A -85,B 0,C 180,E1 -13705.112,E2 -13705.112} C_VEL
LIN {X 0,Y 347.736,Z 262.157,A -85,B 0,C 180,E1 -13709.016,E2 -13709.016} C_VEL
LIN {X 0,Y 347.726,Z 262.155,A -85,B 0,C 180,E1 -13713.073,E2 -13713.073} C_VEL
LIN {X 0,Y 347.764,Z 262.165,A -85,B 0,C 180,E1 -13716.065,E2 -13716.065} C_VEL
LIN {X 0,Y 347.727,Z 262.159,A -85,B 0,C 180,E1 -13718.796,E2 -13718.796} C_VEL
LIN {X 0,Y 347.736,Z 262.169,A -85,B 0,C 180,E1 -13721.832,E2 -13721.832} C_VEL
LIN {X 0,Y 347.698,Z 262.176,A -85,B 0,C 180,E1 -13725.028,E2 -13725.028} C_VEL
LIN {X 0,Y 347.735,Z 262.171,A -85,B 0,C 180,E1 -13728.4,E2 -13728.4} C_VEL
LIN {X 0,Y 347.759,Z 262.151,A -85,B 0,C 180,E1 -13732.014,E2 -13732.014} C_VEL
LIN {X 0,Y 347.81,Z 262.356,A -85,B 0,C 180,E1 -13734.284,E2 -13734.284} C_VEL
LIN {X 0,Y 351.08,Z 275.148,A -85,B 0,C 180,E1 -13737.283,E2 -13737.283} C_VEL
LIN {X 0,Y 353.702,Z 287.071,A -85,B 0,C 180,E1 -13739.895,E2 -13739.895} C_VEL
LIN {X 0,Y 354.159,Z 290.933,A -85,B 0,C 180,E1 -13740.692,E2 -13740.692} C_VEL
LIN {X 0,Y 352.448,Z 306.991,A -85,B 0,C 180,E1 -13743.694,E2 -13743.694} C_VEL
LIN {X 0,Y 351.311,Z 319.1,A -85,B 0,C 180,E1 -13745.893,E2 -13745.893} C_VEL
LIN {X 0,Y 353.802,Z 334.826,A -85,B 0,C 180,E1 -13746.48,E2 -13746.48} C_VEL
LIN {X 0,Y 357.079,Z 358.789,A -85,B 0,C 180,E1 -13747.254,E2 -13747.254} C_VEL
LIN {X 0,Y 358.272,Z 372.133,A -85,B 0,C 180,E1 -13747.632,E2 -13747.632} C_VEL
LIN {X 0,Y 356.997,Z 430.117,A -85,B 0,C 180,E1 -13748.822,E2 -13748.822} C_VEL
LIN {X 0,Y 356.27,Z 443.53,A -85,B 0,C 180,E1 -13749.315,E2 -13749.315} C_VEL
LIN {X 0,Y 354.971,Z 456.787,A -85,B 0,C 180,E1 -13750.03,E2 -13750.03} C_VEL
LIN {X 0,Y 353.652,Z 467.958,A -85,B 0,C 180,E1 -13750.859,E2 -13750.859} C_VEL
LIN {X 0,Y 352.308,Z 478.305,A -85,B 0,C 180,E1 -13751.839,E2 -13751.839} C_VEL
LIN {X 0,Y 350.808,Z 489.046,A -85,B 0,C 180,E1 -13753.113,E2 -13753.113} C_VEL
LIN {X 0,Y 349.448,Z 498.766,A -85,B 0,C 180,E1 -13754.545,E2 -13754.545} C_VEL
LIN {X 0,Y 348.533,Z 506.793,A -85,B 0,C 180,E1 -13755.997,E2 -13755.997} C_VEL
LIN {X 0,Y 347.64,Z 513.472,A -85,B 0,C 180,E1 -13757.448,E2 -13757.448} C_VEL
LIN {X 0,Y 347.027,Z 519.075,A -85,B 0,C 180,E1 -13758.907,E2 -13758.907} C_VEL
LIN {X 0,Y 346.647,Z 524.61,A -85,B 0,C 180,E1 -13760.665,E2 -13760.665} C_VEL
LIN {X 0,Y 346.531,Z 528.978,A -85,B 0,C 180,E1 -13762.425,E2 -13762.425} C_VEL
LIN {X 0,Y 346.674,Z 532.296,A -85,B 0,C 180,E1 -13764.182,E2 -13764.182} C_VEL
LIN {X 0,Y 346.725,Z 533.961,A -85,B 0,C 180,E1 -13765.349,E2 -13765.349} C_VEL
LIN {X 0,Y 346.901,Z 535.209,A -85,B 0,C 180,E1 -13766.515,E2 -13766.515} C_VEL
LIN {X 0,Y 346.964,Z 536.001,A -85,B 0,C 180,E1 -13767.678,E2 -13767.678} C_VEL
LIN {X 0,Y 347.088,Z 536.391,A -85,B 0,C 180,E1 -13770,E2 -13770} C_VEL
LIN {X 0,Y 347.033,Z 535.961,A -85,B 0,C 180,E1 -13771.16,E2 -13771.16} C_VEL
LIN {X 0,Y 347.016,Z 535.085,A -85,B 0,C 180,E1 -13772.321,E2 -13772.321} C_VEL
LIN {X 0,Y 347.064,Z 533.804,A -85,B 0,C 180,E1 -13773.482,E2 -13773.482} C_VEL
LIN {X 0,Y 346.805,Z 531.012,A -85,B 0,C 180,E1 -13775.232,E2 -13775.232} C_VEL
LIN {X 0,Y 346.692,Z 527.168,A -85,B 0,C 180,E1 -13776.986,E2 -13776.986} C_VEL
LIN {X 0,Y 346.695,Z 522.166,A -85,B 0,C 180,E1 -13778.744,E2 -13778.744} C_VEL
LIN {X 0,Y 346.898,Z 515.866,A -85,B 0,C 180,E1 -13780.505,E2 -13780.505} C_VEL
LIN {X 0,Y 347.395,Z 508.05,A -85,B 0,C 180,E1 -13782.263,E2 -13782.263} C_VEL
LIN {X 0,Y 348.099,Z 500.07,A -85,B 0,C 180,E1 -13783.722,E2 -13783.722} C_VEL
LIN {X 0,Y 348.871,Z 491.433,A -85,B 0,C 180,E1 -13785.029,E2 -13785.029} C_VEL
LIN {X 0,Y 349.891,Z 480.858,A -85,B 0,C 180,E1 -13786.331,E2 -13786.331} C_VEL
LIN {X 0,Y 350.998,Z 469.156,A -85,B 0,C 180,E1 -13787.477,E2 -13787.477} C_VEL
LIN {X 0,Y 352.145,Z 456.835,A -85,B 0,C 180,E1 -13788.395,E2 -13788.395} C_VEL
LIN {X 0,Y 353.062,Z 443.082,A -85,B 0,C 180,E1 -13789.136,E2 -13789.136} C_VEL
LIN {X 0,Y 353.632,Z 430.058,A -85,B 0,C 180,E1 -13789.594,E2 -13789.594} C_VEL
LIN {X 0,Y 354.51,Z 369.681,A -85,B 0,C 180,E1 -13790.825,E2 -13790.825} C_VEL
LIN {X 0,Y 349.518,Z 320.346,A -85,B 0,C 180,E1 -13792.148,E2 -13792.148} C_VEL
LIN {X 0,Y 351.29,Z 296.652,A -85,B 0,C 180,E1 -13796.431,E2 -13796.431} C_VEL
LIN {X 0,Y 352.239,Z 284.729,A -85,B 0,C 180,E1 -13798.609,E2 -13798.609} C_VEL
LIN {X 0,Y 350.841,Z 276.402,A -85,B 0,C 180,E1 -13800.264,E2 -13800.264} C_VEL
LIN {X 0,Y 347.907,Z 262.946,A -85,B 0,C 180,E1 -13803.052,E2 -13803.052} C_VEL
LIN {X 0,Y 347.762,Z 262.216,A -85,B 0,C 180,E1 -13803.311,E2 -13803.311} C_VEL
LIN {X 0,Y 347.76,Z 262.164,A -85,B 0,C 180,E1 -13806.063,E2 -13806.063} C_VEL
LIN {X 0,Y 347.725,Z 262.169,A -85,B 0,C 180,E1 -13808.795,E2 -13808.795} C_VEL
LIN {X 0,Y 347.733,Z 262.168,A -85,B 0,C 180,E1 -13811.831,E2 -13811.831} C_VEL
LIN {X 0,Y 347.693,Z 262.173,A -85,B 0,C 180,E1 -13815.027,E2 -13815.027} C_VEL
LIN {X 0,Y 347.73,Z 262.167,A -85,B 0,C 180,E1 -13818.399,E2 -13818.399} C_VEL
LIN {X 0,Y 347.753,Z 262.163,A -85,B 0,C 180,E1 -13822.013,E2 -13822.013} C_VEL
LIN {X 0,Y 347.734,Z 262.168,A -85,B 0,C 180,E1 -13825.535,E2 -13825.535} C_VEL
LIN {X 0,Y 347.72,Z 262.167,A -85,B 0,C 180,E1 -13828.298,E2 -13828.298} C_VEL
LIN {X 0,Y 347.731,Z 262.173,A -85,B 0,C 180,E1 -13830.983,E2 -13830.983} C_VEL
LIN {X 0,Y 347.756,Z 262.168,A -85,B 0,C 180,E1 -13834.887,E2 -13834.887} C_VEL
LIN {X 0,Y 347.768,Z 262.166,A -85,B 0,C 180,E1 -13838.669,E2 -13838.669} C_VEL
LIN {X 0,Y 347.832,Z 262.155,A -85,B 0,C 180,E1 -13842.358,E2 -13842.358} C_VEL
LIN {X 0,Y 347.888,Z 262.148,A -85,B 0,C 180,E1 -13845.971,E2 -13845.971} C_VEL
LIN {X 0,Y 347.881,Z 262.147,A -85,B 0,C 180,E1 -13849.524,E2 -13849.524} C_VEL
LIN {X 0,Y 348.038,Z 262.131,A -85,B 0,C 180,E1 -13853.041,E2 -13853.041} C_VEL
LIN {X 0,Y 348.179,Z 262.11,A -85,B 0,C 180,E1 -13857.687,E2 -13857.687} C_VEL
LIN {X 0,Y 348.127,Z 262.117,A -85,B 0,C 180,E1 -13861.157,E2 -13861.157} C_VEL
LIN {X 0,Y 348.167,Z 262.116,A -85,B 0,C 180,E1 -13862.314,E2 -13862.314} C_VEL
LIN {X 0,Y 348.04,Z 262.128,A -85,B 0,C 180,E1 -13866.959,E2 -13866.959} C_VEL
LIN {X 0,Y 347.879,Z 262.153,A -85,B 0,C 180,E1 -13870.476,E2 -13870.476} C_VEL
LIN {X 0,Y 347.889,Z 262.152,A -85,B 0,C 180,E1 -13874.151,E2 -13874.151} C_VEL
LIN {X 0,Y 347.82,Z 262.16,A -85,B 0,C 180,E1 -13878.26,E2 -13878.26} C_VEL
LIN {X 0,Y 347.757,Z 262.165,A -85,B 0,C 180,E1 -13881.626,E2 -13881.626} C_VEL
LIN {X 0,Y 347.729,Z 262.166,A -85,B 0,C 180,E1 -13885.115,E2 -13885.115} C_VEL
LIN {X 0,Y 347.716,Z 262.17,A -85,B 0,C 180,E1 -13887.702,E2 -13887.702} C_VEL
LIN {X 0,Y 347.728,Z 262.17,A -85,B 0,C 180,E1 -13890.35,E2 -13890.35} C_VEL
LIN {X 0,Y 347.741,Z 262.17,A -85,B 0,C 180,E1 -13894.045,E2 -13894.045} C_VEL
LIN {X 0,Y 347.747,Z 262.166,A -85,B 0,C 180,E1 -13897.323,E2 -13897.323} C_VEL
LIN {X 0,Y 347.69,Z 262.172,A -85,B 0,C 180,E1 -13900.304,E2 -13900.304} C_VEL
LIN {X 0,Y 347.715,Z 262.166,A -85,B 0,C 180,E1 -13903.41,E2 -13903.41} C_VEL
LIN {X 0,Y 347.718,Z 262.168,A -85,B 0,C 180,E1 -13906.688,E2 -13906.688} C_VEL
LIN {X 0,Y 347.697,Z 262.172,A -85,B 0,C 180,E1 -13910.184,E2 -13910.184} C_VEL
LIN {X 0,Y 347.751,Z 262.16,A -85,B 0,C 180,E1 -13912.679,E2 -13912.679} C_VEL
LIN {X 0,Y 347.746,Z 262.168,A -85,B 0,C 180,E1 -13915.958,E2 -13915.958} C_VEL
LIN {X 0,Y 347.725,Z 262.171,A -85,B 0,C 180,E1 -13919.651,E2 -13919.651} C_VEL
LIN {X 0,Y 347.734,Z 262.17,A -85,B 0,C 180,E1 -13923.601,E2 -13923.601} C_VEL
LIN {X 0,Y 347.751,Z 262.165,A -85,B 0,C 180,E1 -13926.16,E2 -13926.16} C_VEL
LIN {X 0,Y 347.743,Z 262.162,A -85,B 0,C 180,E1 -13929.906,E2 -13929.906} C_VEL
LIN {X 0,Y 347.809,Z 262.157,A -85,B 0,C 180,E1 -13932.357,E2 -13932.357} C_VEL
LIN {X 0,Y 347.878,Z 262.288,A -85,B 0,C 180,E1 -13936.137,E2 -13936.137} C_VEL
LIN {X 0,Y 348.088,Z 263.203,A -85,B 0,C 180,E1 -13936.342,E2 -13936.342} C_VEL
LIN {X 0,Y 355.681,Z 283.022,A -85,B 0,C 180,E1 -13937.219,E2 -13937.219} C_VEL
LIN {X 0,Y 354.684,Z 349.436,A -85,B 0,C 180,E1 -13938.572,E2 -13938.572} C_VEL
LIN {X 0,Y 354.453,Z 362.614,A -85,B 0,C 180,E1 -13939.071,E2 -13939.071} C_VEL
LIN {X 0,Y 354.076,Z 375.199,A -85,B 0,C 180,E1 -13939.782,E2 -13939.782} C_VEL
LIN {X 0,Y 353.363,Z 387.267,A -85,B 0,C 180,E1 -13940.701,E2 -13940.701} C_VEL
LIN {X 0,Y 352.492,Z 398.672,A -85,B 0,C 180,E1 -13941.834,E2 -13941.834} C_VEL
LIN {X 0,Y 351.658,Z 408.924,A -85,B 0,C 180,E1 -13943.114,E2 -13943.114} C_VEL
LIN {X 0,Y 350.838,Z 418.169,A -85,B 0,C 180,E1 -13944.541,E2 -13944.541} C_VEL
LIN {X 0,Y 349.944,Z 427.087,A -85,B 0,C 180,E1 -13946.258,E2 -13946.258} C_VEL
LIN {X 0,Y 349.087,Z 434.303,A -85,B 0,C 180,E1 -13947.981,E2 -13947.981} C_VEL
LIN {X 0,Y 348.47,Z 440.9,A -85,B 0,C 180,E1 -13950,E2 -13950} C_VEL
LIN {X 0,Y 347.99,Z 445.279,A -85,B 0,C 180,E1 -13951.736,E2 -13951.736} C_VEL
LIN {X 0,Y 347.599,Z 448.616,A -85,B 0,C 180,E1 -13953.478,E2 -13953.478} C_VEL
LIN {X 0,Y 347.576,Z 450.258,A -85,B 0,C 180,E1 -13954.64,E2 -13954.64} C_VEL
LIN {X 0,Y 347.529,Z 451.519,A -85,B 0,C 180,E1 -13955.804,E2 -13955.804} C_VEL
LIN {X 0,Y 347.485,Z 452.71,A -85,B 0,C 180,E1 -13957.671,E2 -13957.671} C_VEL
LIN {X 0,Y 347.551,Z 452.921,A -85,B 0,C 180,E1 -13959.31,E2 -13959.31} C_VEL
LIN {X 0,Y 347.809,Z 451.917,A -85,B 0,C 180,E1 -13961.658,E2 -13961.658} C_VEL
LIN {X 0,Y 348.034,Z 450.776,A -85,B 0,C 180,E1 -13962.834,E2 -13962.834} C_VEL
LIN {X 0,Y 348.592,Z 448.305,A -85,B 0,C 180,E1 -13964.592,E2 -13964.592} C_VEL
LIN {X 0,Y 349.204,Z 444.806,A -85,B 0,C 180,E1 -13966.365,E2 -13966.365} C_VEL
LIN {X 0,Y 350.008,Z 440.179,A -85,B 0,C 180,E1 -13968.134,E2 -13968.134} C_VEL
LIN {X 0,Y 351.211,Z 433.157,A -85,B 0,C 180,E1 -13970.193,E2 -13970.193} C_VEL
LIN {X 0,Y 352.457,Z 425.436,A -85,B 0,C 180,E1 -13971.955,E2 -13971.955} C_VEL
LIN {X 0,Y 353.86,Z 416.024,A -85,B 0,C 180,E1 -13973.656,E2 -13973.656} C_VEL
LIN {X 0,Y 354.965,Z 406.613,A -85,B 0,C 180,E1 -13975.037,E2 -13975.037} C_VEL
LIN {X 0,Y 356.102,Z 396.666,A -85,B 0,C 180,E1 -13976.205,E2 -13976.205} C_VEL
LIN {X 0,Y 357.15,Z 385.831,A -85,B 0,C 180,E1 -13977.22,E2 -13977.22} C_VEL
LIN {X 0,Y 357.875,Z 375.792,A -85,B 0,C 180,E1 -13977.969,E2 -13977.969} C_VEL
LIN {X 0,Y 358.455,Z 362.618,A -85,B 0,C 180,E1 -13978.708,E2 -13978.708} C_VEL
LIN {X 0,Y 358.711,Z 350.533,A -85,B 0,C 180,E1 -13979.167,E2 -13979.167} C_VEL
LIN {X 0,Y 359.093,Z 320.207,A -85,B 0,C 180,E1 -13979.824,E2 -13979.824} C_VEL
LIN {X 0,Y 358.682,Z 310.405,A -85,B 0,C 180,E1 -13980.07,E2 -13980.07} C_VEL
LIN {X 0,Y 357.814,Z 304.63,A -85,B 0,C 180,E1 -13980.265,E2 -13980.265} C_VEL
LIN {X 0,Y 355.987,Z 297.129,A -85,B 0,C 180,E1 -13980.574,E2 -13980.574} C_VEL
LIN {X 0,Y 353.432,Z 289.942,A -85,B 0,C 180,E1 -13980.94,E2 -13980.94} C_VEL
LIN {X 0,Y 345.119,Z 272.334,A -85,B 0,C 180,E1 -13982.042,E2 -13982.042} C_VEL
LIN {X 0,Y 340.896,Z 264.003,A -85,B 0,C 180,E1 -13982.641,E2 -13982.641} C_VEL
LIN {X 0,Y 340.703,Z 263.121,A -85,B 0,C 180,E1 -13982.89,E2 -13982.89} C_VEL
LIN {X 0,Y 340.708,Z 262.997,A -85,B 0,C 180,E1 -13986.439,E2 -13986.439} C_VEL
LIN {X 0,Y 340.655,Z 263.054,A -85,B 0,C 180,E1 -13989.758,E2 -13989.758} C_VEL
LIN {X 0,Y 340.672,Z 263.041,A -85,B 0,C 180,E1 -13992.904,E2 -13992.904} C_VEL
LIN {X 0,Y 340.671,Z 263.031,A -85,B 0,C 180,E1 -13997.094,E2 -13997.094} C_VEL
LIN {X 0,Y 340.653,Z 263.049,A -85,B 0,C 180,E1 -14000.24,E2 -14000.24} C_VEL
LIN {X 0,Y 340.706,Z 263.027,A -85,B 0,C 180,E1 -14003.559,E2 -14003.559} C_VEL
LIN {X 0,Y 340.691,Z 263.051,A -85,B 0,C 180,E1 -14006.153,E2 -14006.153} C_VEL
LIN {X 0,Y 340.719,Z 263.011,A -85,B 0,C 180,E1 -14010.034,E2 -14010.034} C_VEL
LIN {X 0,Y 340.715,Z 263.044,A -85,B 0,C 180,E1 -14013.012,E2 -14013.012} C_VEL
LIN {X 0,Y 340.741,Z 263.028,A -85,B 0,C 180,E1 -14015.637,E2 -14015.637} C_VEL
LIN {X 0,Y 340.729,Z 263.011,A -85,B 0,C 180,E1 -14019.473,E2 -14019.473} C_VEL
LIN {X 0,Y 340.854,Z 263.024,A -85,B 0,C 180,E1 -14021.984,E2 -14021.984} C_VEL
LIN {X 0,Y 340.866,Z 263.014,A -85,B 0,C 180,E1 -14025.705,E2 -14025.705} C_VEL
LIN {X 0,Y 340.842,Z 263.026,A -85,B 0,C 180,E1 -14029.305,E2 -14029.305} C_VEL
LIN {X 0,Y 340.994,Z 263.007,A -85,B 0,C 180,E1 -14032.896,E2 -14032.896} C_VEL
LIN {X 0,Y 340.802,Z 263.026,A -85,B 0,C 180,E1 -14035.268,E2 -14035.268} C_VEL
LIN {X 0,Y 341.117,Z 262.988,A -85,B 0,C 180,E1 -14037.638,E2 -14037.638} C_VEL
LIN {X 0,Y 341.082,Z 262.989,A -85,B 0,C 180,E1 -14041.18,E2 -14041.18} C_VEL
LIN {X 0,Y 341.123,Z 262.982,A -85,B 0,C 180,E1 -14042.361,E2 -14042.361} C_VEL
LIN {X 0,Y 340.991,Z 262.998,A -85,B 0,C 180,E1 -14047.103,E2 -14047.103} C_VEL
LIN {X 0,Y 340.841,Z 263.027,A -85,B 0,C 180,E1 -14050.695,E2 -14050.695} C_VEL
LIN {X 0,Y 340.859,Z 263.021,A -85,B 0,C 180,E1 -14054.325,E2 -14054.325} C_VEL
LIN {X 0,Y 340.782,Z 263.028,A -85,B 0,C 180,E1 -14058.44,E2 -14058.44} C_VEL
LIN {X 0,Y 340.714,Z 263.037,A -85,B 0,C 180,E1 -14061.842,E2 -14061.842} C_VEL
LIN {X 0,Y 340.71,Z 263.036,A -85,B 0,C 180,E1 -14065.669,E2 -14065.669} C_VEL
LIN {X 0,Y 340.697,Z 263.043,A -85,B 0,C 180,E1 -14069.675,E2 -14069.675} C_VEL
LIN {X 0,Y 340.677,Z 263.041,A -85,B 0,C 180,E1 -14072.437,E2 -14072.437} C_VEL
LIN {X 0,Y 340.713,Z 263.038,A -85,B 0,C 180,E1 -14075.279,E2 -14075.279} C_VEL
LIN {X 0,Y 340.689,Z 263.037,A -85,B 0,C 180,E1 -14078.382,E2 -14078.382} C_VEL
LIN {X 0,Y 340.687,Z 263.047,A -85,B 0,C 180,E1 -14082.044,E2 -14082.044} C_VEL
LIN {X 0,Y 340.647,Z 263.046,A -85,B 0,C 180,E1 -14086.228,E2 -14086.228} C_VEL
LIN {X 0,Y 340.666,Z 263.047,A -85,B 0,C 180,E1 -14088.688,E2 -14088.688} C_VEL
LIN {X 0,Y 340.716,Z 263.024,A -85,B 0,C 180,E1 -14091.771,E2 -14091.771} C_VEL
LIN {X 0,Y 340.737,Z 263.246,A -85,B 0,C 180,E1 -14093.752,E2 -14093.752} C_VEL
LIN {X 0,Y 344.13,Z 276.102,A -85,B 0,C 180,E1 -14096.859,E2 -14096.859} C_VEL
LIN {X 0,Y 346.737,Z 288.114,A -85,B 0,C 180,E1 -14099.554,E2 -14099.554} C_VEL
LIN {X 0,Y 347.375,Z 292.33,A -85,B 0,C 180,E1 -14100.455,E2 -14100.455} C_VEL
LIN {X 0,Y 345.567,Z 308.265,A -85,B 0,C 180,E1 -14103.49,E2 -14103.49} C_VEL
LIN {X 0,Y 344.609,Z 318.12,A -85,B 0,C 180,E1 -14105.315,E2 -14105.315} C_VEL
LIN {X 0,Y 346.28,Z 328.587,A -85,B 0,C 180,E1 -14105.74,E2 -14105.74} C_VEL
LIN {X 0,Y 350.012,Z 354.271,A -85,B 0,C 180,E1 -14106.619,E2 -14106.619} C_VEL
LIN {X 0,Y 351.811,Z 372.223,A -85,B 0,C 180,E1 -14107.156,E2 -14107.156} C_VEL
LIN {X 0,Y 350.478,Z 429.824,A -85,B 0,C 180,E1 -14108.364,E2 -14108.364} C_VEL
LIN {X 0,Y 349.658,Z 443.916,A -85,B 0,C 180,E1 -14108.905,E2 -14108.905} C_VEL
LIN {X 0,Y 348.305,Z 456.767,A -85,B 0,C 180,E1 -14109.631,E2 -14109.631} C_VEL
LIN {X 0,Y 346.708,Z 469.323,A -85,B 0,C 180,E1 -14110.614,E2 -14110.614} C_VEL
LIN {X 0,Y 345.188,Z 480.562,A -85,B 0,C 180,E1 -14111.758,E2 -14111.758} C_VEL
LIN {X 0,Y 343.674,Z 490.724,A -85,B 0,C 180,E1 -14113.058,E2 -14113.058} C_VEL
LIN {X 0,Y 342.331,Z 499.946,A -85,B 0,C 180,E1 -14114.521,E2 -14114.521} C_VEL
LIN {X 0,Y 341.187,Z 508.997,A -85,B 0,C 180,E1 -14116.297,E2 -14116.297} C_VEL
LIN {X 0,Y 340.25,Z 516.324,A -85,B 0,C 180,E1 -14118.079,E2 -14118.079} C_VEL
LIN {X 0,Y 339.665,Z 522.226,A -85,B 0,C 180,E1 -14119.87,E2 -14119.87} C_VEL
LIN {X 0,Y 339.499,Z 526.937,A -85,B 0,C 180,E1 -14121.668,E2 -14121.668} C_VEL
LIN {X 0,Y 339.57,Z 530.521,A -85,B 0,C 180,E1 -14123.437,E2 -14123.437} C_VEL
LIN {X 0,Y 339.641,Z 533.174,A -85,B 0,C 180,E1 -14125.252,E2 -14125.252} C_VEL
LIN {X 0,Y 339.828,Z 534.393,A -85,B 0,C 180,E1 -14126.442,E2 -14126.442} C_VEL
LIN {X 0,Y 339.914,Z 535.173,A -85,B 0,C 180,E1 -14127.63,E2 -14127.63} C_VEL
LIN {X 0,Y 340.039,Z 535.533,A -85,B 0,C 180,E1 -14130,E2 -14130} C_VEL
LIN {X 0,Y 339.983,Z 535.075,A -85,B 0,C 180,E1 -14131.184,E2 -14131.184} C_VEL
LIN {X 0,Y 339.969,Z 534.181,A -85,B 0,C 180,E1 -14132.369,E2 -14132.369} C_VEL
LIN {X 0,Y 340,Z 532.882,A -85,B 0,C 180,E1 -14133.555,E2 -14133.555} C_VEL
LIN {X 0,Y 339.732,Z 530.053,A -85,B 0,C 180,E1 -14135.341,E2 -14135.341} C_VEL
LIN {X 0,Y 339.625,Z 526.173,A -85,B 0,C 180,E1 -14137.132,E2 -14137.132} C_VEL
LIN {X 0,Y 339.63,Z 521.129,A -85,B 0,C 180,E1 -14138.928,E2 -14138.928} C_VEL
LIN {X 0,Y 339.847,Z 514.783,A -85,B 0,C 180,E1 -14140.726,E2 -14140.726} C_VEL
LIN {X 0,Y 340.387,Z 506.902,A -85,B 0,C 180,E1 -14142.52,E2 -14142.52} C_VEL
LIN {X 0,Y 341.089,Z 498.845,A -85,B 0,C 180,E1 -14144.01,E2 -14144.01} C_VEL
LIN {X 0,Y 342.101,Z 489.044,A -85,B 0,C 180,E1 -14145.489,E2 -14145.489} C_VEL
LIN {X 0,Y 343.015,Z 479.476,A -85,B 0,C 180,E1 -14146.668,E2 -14146.668} C_VEL
LIN {X 0,Y 344.179,Z 467.653,A -85,B 0,C 180,E1 -14147.835,E2 -14147.835} C_VEL
LIN {X 0,Y 345.368,Z 455.062,A -85,B 0,C 180,E1 -14148.769,E2 -14148.769} C_VEL
LIN {X 0,Y 346.301,Z 441.767,A -85,B 0,C 180,E1 -14149.486,E2 -14149.486} C_VEL
LIN {X 0,Y 346.826,Z 429.746,A -85,B 0,C 180,E1 -14149.918,E2 -14149.918} C_VEL
LIN {X 0,Y 347.659,Z 369.148,A -85,B 0,C 180,E1 -14151.184,E2 -14151.184} C_VEL
LIN {X 0,Y 342.593,Z 319.647,A -85,B 0,C 180,E1 -14152.535,E2 -14152.535} C_VEL
LIN {X 0,Y 344.534,Z 295.42,A -85,B 0,C 180,E1 -14156.991,E2 -14156.991} C_VEL
LIN {X 0,Y 345.248,Z 285.143,A -85,B 0,C 180,E1 -14158.917,E2 -14158.917} C_VEL
LIN {X 0,Y 342.826,Z 272.516,A -85,B 0,C 180,E1 -14161.515,E2 -14161.515} C_VEL
LIN {X 0,Y 340.728,Z 263.142,A -85,B 0,C 180,E1 -14163.575,E2 -14163.575} C_VEL
LIN {X 0,Y 340.695,Z 263.044,A -85,B 0,C 180,E1 -14166.741,E2 -14166.741} C_VEL
LIN {X 0,Y 340.644,Z 263.049,A -85,B 0,C 180,E1 -14170.238,E2 -14170.238} C_VEL
LIN {X 0,Y 340.665,Z 263.05,A -85,B 0,C 180,E1 -14172.904,E2 -14172.904} C_VEL
LIN {X 0,Y 340.664,Z 263.049,A -85,B 0,C 180,E1 -14177.094,E2 -14177.094} C_VEL
LIN {X 0,Y 340.647,Z 263.049,A -85,B 0,C 180,E1 -14180.24,E2 -14180.24} C_VEL
LIN {X 0,Y 340.698,Z 263.045,A -85,B 0,C 180,E1 -14183.56,E2 -14183.56} C_VEL
LIN {X 0,Y 340.681,Z 263.044,A -85,B 0,C 180,E1 -14186.152,E2 -14186.152} C_VEL
LIN {X 0,Y 340.707,Z 263.041,A -85,B 0,C 180,E1 -14190.035,E2 -14190.035} C_VEL
LIN {X 0,Y 340.7,Z 263.047,A -85,B 0,C 180,E1 -14193.011,E2 -14193.011} C_VEL
LIN {X 0,Y 340.729,Z 263.039,A -85,B 0,C 180,E1 -14195.636,E2 -14195.636} C_VEL
LIN {X 0,Y 340.706,Z 263.042,A -85,B 0,C 180,E1 -14199.472,E2 -14199.472} C_VEL
LIN {X 0,Y 340.781,Z 263.03,A -85,B 0,C 180,E1 -14201.98,E2 -14201.98} C_VEL
LIN {X 0,Y 340.842,Z 263.025,A -85,B 0,C 180,E1 -14205.716,E2 -14205.716} C_VEL
LIN {X 0,Y 340.834,Z 263.025,A -85,B 0,C 180,E1 -14209.305,E2 -14209.305} C_VEL
LIN {X 0,Y 340.986,Z 263.01,A -85,B 0,C 180,E1 -14212.897,E2 -14212.897} C_VEL
LIN {X 0,Y 340.802,Z 263.03,A -85,B 0,C 180,E1 -14215.269,E2 -14215.269} C_VEL
LIN {X 0,Y 341.116,Z 262.99,A -85,B 0,C 180,E1 -14217.639,E2 -14217.639} C_VEL
LIN {X 0,Y 341.096,Z 262.993,A -85,B 0,C 180,E1 -14221.181,E2 -14221.181} C_VEL
LIN {X 0,Y 341.104,Z 262.996,A -85,B 0,C 180,E1 -14222.362,E2 -14222.362} C_VEL
LIN {X 0,Y 340.974,Z 263.006,A -85,B 0,C 180,E1 -14226.599,E2 -14226.599} C_VEL
LIN {X 0,Y 340.869,Z 263.019,A -85,B 0,C 180,E1 -14229.494,E2 -14229.494} C_VEL
LIN {X 0,Y 340.831,Z 263.026,A -85,B 0,C 180,E1 -14233.11,E2 -14233.11} C_VEL
LIN {X 0,Y 340.806,Z 263.029,A -85,B 0,C 180,E1 -14235.551,E2 -14235.551} C_VEL
LIN {X 0,Y 340.725,Z 263.038,A -85,B 0,C 180,E1 -14239.271,E2 -14239.271} C_VEL
LIN {X 0,Y 340.695,Z 263.043,A -85,B 0,C 180,E1 -14243.076,E2 -14243.076} C_VEL
LIN {X 0,Y 340.702,Z 263.041,A -85,B 0,C 180,E1 -14246.989,E2 -14246.989} C_VEL
LIN {X 0,Y 340.684,Z 263.044,A -85,B 0,C 180,E1 -14251.047,E2 -14251.047} C_VEL
LIN {X 0,Y 340.708,Z 263.042,A -85,B 0,C 180,E1 -14255.281,E2 -14255.281} C_VEL
LIN {X 0,Y 340.686,Z 263.045,A -85,B 0,C 180,E1 -14258.383,E2 -14258.383} C_VEL
LIN {X 0,Y 340.685,Z 263.041,A -85,B 0,C 180,E1 -14262.045,E2 -14262.045} C_VEL
LIN {X 0,Y 340.644,Z 263.051,A -85,B 0,C 180,E1 -14266.229,E2 -14266.229} C_VEL
LIN {X 0,Y 340.664,Z 263.047,A -85,B 0,C 180,E1 -14268.689,E2 -14268.689} C_VEL
LIN {X 0,Y 340.715,Z 263.04,A -85,B 0,C 180,E1 -14271.772,E2 -14271.772} C_VEL
LIN {X 0,Y 340.72,Z 263.045,A -85,B 0,C 180,E1 -14275.597,E2 -14275.597} C_VEL
LIN {X 0,Y 340.679,Z 263.045,A -85,B 0,C 180,E1 -14278.955,E2 -14278.955} C_VEL
LIN {X 0,Y 340.709,Z 263.044,A -85,B 0,C 180,E1 -14283.013,E2 -14283.013} C_VEL
LIN {X 0,Y 340.704,Z 263.044,A -85,B 0,C 180,E1 -14286.927,E2 -14286.927} C_VEL
LIN {X 0,Y 340.694,Z 263.037,A -85,B 0,C 180,E1 -14290.729,E2 -14290.729} C_VEL
LIN {X 0,Y 340.738,Z 263.043,A -85,B 0,C 180,E1 -14293.217,E2 -14293.217} C_VEL
LIN {X 0,Y 340.845,Z 263.283,A -85,B 0,C 180,E1 -14295.776,E2 -14295.776} C_VEL
LIN {X 0,Y 341.13,Z 264.391,A -85,B 0,C 180,E1 -14295.958,E2 -14295.958} C_VEL
LIN {X 0,Y 347.53,Z 280.69,A -85,B 0,C 180,E1 -14296.712,E2 -14296.712} C_VEL
LIN {X 0,Y 348.853,Z 284.346,A -85,B 0,C 180,E1 -14296.866,E2 -14296.866} C_VEL
LIN {X 0,Y 347.92,Z 351.161,A -85,B 0,C 180,E1 -14298.268,E2 -14298.268} C_VEL
LIN {X 0,Y 347.639,Z 364.139,A -85,B 0,C 180,E1 -14298.78,E2 -14298.78} C_VEL
LIN {X 0,Y 347.253,Z 376.543,A -85,B 0,C 180,E1 -14299.506,E2 -14299.506} C_VEL
LIN {X 0,Y 346.573,Z 387.676,A -85,B 0,C 180,E1 -14300.37,E2 -14300.37} C_VEL
LIN {X 0,Y 345.667,Z 399.167,A -85,B 0,C 180,E1 -14301.524,E2 -14301.524} C_VEL
LIN {X 0,Y 344.8,Z 409.479,A -85,B 0,C 180,E1 -14302.829,E2 -14302.829} C_VEL
LIN {X 0,Y 344.023,Z 417.915,A -85,B 0,C 180,E1 -14304.138,E2 -14304.138} C_VEL
LIN {X 0,Y 343.231,Z 425.701,A -85,B 0,C 180,E1 -14305.597,E2 -14305.597} C_VEL
LIN {X 0,Y 342.328,Z 433.348,A -85,B 0,C 180,E1 -14307.353,E2 -14307.353} C_VEL
LIN {X 0,Y 341.724,Z 438.56,A -85,B 0,C 180,E1 -14308.822,E2 -14308.822} C_VEL
LIN {X 0,Y 341.202,Z 443.627,A -85,B 0,C 180,E1 -14310.591,E2 -14310.591} C_VEL
LIN {X 0,Y 340.764,Z 447.58,A -85,B 0,C 180,E1 -14312.364,E2 -14312.364} C_VEL
LIN {X 0,Y 340.546,Z 449.625,A -85,B 0,C 180,E1 -14313.55,E2 -14313.55} C_VEL
LIN {X 0,Y 340.536,Z 451.236,A -85,B 0,C 180,E1 -14314.736,E2 -14314.736} C_VEL
LIN {X 0,Y 340.485,Z 452.47,A -85,B 0,C 180,E1 -14315.924,E2 -14315.924} C_VEL
LIN {X 0,Y 340.437,Z 453.561,A -85,B 0,C 180,E1 -14317.724,E2 -14317.724} C_VEL
LIN {X 0,Y 340.526,Z 453.76,A -85,B 0,C 180,E1 -14319.504,E2 -14319.504} C_VEL
LIN {X 0,Y 340.644,Z 453.423,A -85,B 0,C 180,E1 -14320.701,E2 -14320.701} C_VEL
LIN {X 0,Y 340.822,Z 452.676,A -85,B 0,C 180,E1 -14321.9,E2 -14321.9} C_VEL
LIN {X 0,Y 341.079,Z 451.5,A -85,B 0,C 180,E1 -14323.101,E2 -14323.101} C_VEL
LIN {X 0,Y 341.64,Z 449.147,A -85,B 0,C 180,E1 -14324.791,E2 -14324.791} C_VEL
LIN {X 0,Y 342.344,Z 445.404,A -85,B 0,C 180,E1 -14326.703,E2 -14326.703} C_VEL
LIN {X 0,Y 343.196,Z 440.709,A -85,B 0,C 180,E1 -14328.506,E2 -14328.506} C_VEL
LIN {X 0,Y 344.276,Z 434.719,A -85,B 0,C 180,E1 -14330.306,E2 -14330.306} C_VEL
LIN {X 0,Y 345.585,Z 427.208,A -85,B 0,C 180,E1 -14332.1,E2 -14332.1} C_VEL
LIN {X 0,Y 346.773,Z 419.462,A -85,B 0,C 180,E1 -14333.595,E2 -14333.595} C_VEL
LIN {X 0,Y 348.031,Z 409.917,A -85,B 0,C 180,E1 -14335.091,E2 -14335.091} C_VEL
LIN {X 0,Y 349.389,Z 399.239,A -85,B 0,C 180,E1 -14336.426,E2 -14336.426} C_VEL
LIN {X 0,Y 350.427,Z 388.843,A -85,B 0,C 180,E1 -14337.469,E2 -14337.469} C_VEL
LIN {X 0,Y 351.37,Z 376.869,A -85,B 0,C 180,E1 -14338.4,E2 -14338.4} C_VEL
LIN {X 0,Y 352.003,Z 363.57,A -85,B 0,C 180,E1 -14339.162,E2 -14339.162} C_VEL
LIN {X 0,Y 352.285,Z 351.545,A -85,B 0,C 180,E1 -14339.629,E2 -14339.629} C_VEL
LIN {X 0,Y 352.994,Z 310.793,A -85,B 0,C 180,E1 -14340.508,E2 -14340.508} C_VEL
LIN {X 0,Y 353.432,Z 289.942,A -85,B 0,C 180,E1 -14340.94,E2 -14340.94} C_VEL
LIN {X 0,Y 351.414,Z 286.856,A -85,B 0,C 180,E1 -14341.175,E2 -14341.175} C_VEL
LIN {X 0,Y 346.714,Z 283.039,A -85,B 0,C 180,E1 -14341.657,E2 -14341.657} C_VEL
LIN {X 0,Y 341.909,Z 279.312,A -85,B 0,C 180,E1 -14342.161,E2 -14342.161} C_VEL
LIN {X 0,Y 339.726,Z 276.34,A -85,B 0,C 180,E1 -14342.426,E2 -14342.426} C_VEL
LIN {X 0,Y 333.864,Z 264.882,A -85,B 0,C 180,E1 -14343.276,E2 -14343.276} C_VEL
LIN {X 0,Y 333.676,Z 263.987,A -85,B 0,C 180,E1 -14343.542,E2 -14343.542} C_VEL
LIN {X 0,Y 333.662,Z 263.874,A -85,B 0,C 180,E1 -14346.831,E2 -14346.831} C_VEL
LIN {X 0,Y 333.603,Z 263.926,A -85,B 0,C 180,E1 -14350.773,E2 -14350.773} C_VEL
LIN {X 0,Y 333.59,Z 263.936,A -85,B 0,C 180,E1 -14354.249,E2 -14354.249} C_VEL
LIN {X 0,Y 333.634,Z 263.91,A -85,B 0,C 180,E1 -14357.617,E2 -14357.617} C_VEL
LIN {X 0,Y 333.614,Z 263.914,A -85,B 0,C 180,E1 -14361.21,E2 -14361.21} C_VEL
LIN {X 0,Y 333.673,Z 263.907,A -85,B 0,C 180,E1 -14363.86,E2 -14363.86} C_VEL
LIN {X 0,Y 333.642,Z 263.917,A -85,B 0,C 180,E1 -14367.413,E2 -14367.413} C_VEL
LIN {X 0,Y 333.65,Z 263.902,A -85,B 0,C 180,E1 -14371.022,E2 -14371.022} C_VEL
LIN {X 0,Y 333.694,Z 263.914,A -85,B 0,C 180,E1 -14375.088,E2 -14375.088} C_VEL
LIN {X 0,Y 333.661,Z 263.884,A -85,B 0,C 180,E1 -14379.018,E2 -14379.018} C_VEL
LIN {X 0,Y 333.79,Z 263.9,A -85,B 0,C 180,E1 -14381.589,E2 -14381.589} C_VEL
LIN {X 0,Y 333.805,Z 263.893,A -85,B 0,C 180,E1 -14385.576,E2 -14385.576} C_VEL
LIN {X 0,Y 333.812,Z 263.901,A -85,B 0,C 180,E1 -14389.077,E2 -14389.077} C_VEL
LIN {X 0,Y 333.95,Z 263.884,A -85,B 0,C 180,E1 -14392.746,E2 -14392.746} C_VEL
LIN {X 0,Y 333.769,Z 263.903,A -85,B 0,C 180,E1 -14395.168,E2 -14395.168} C_VEL
LIN {X 0,Y 334.058,Z 263.866,A -85,B 0,C 180,E1 -14397.588,E2 -14397.588} C_VEL
LIN {X 0,Y 334.053,Z 263.864,A -85,B 0,C 180,E1 -14401.205,E2 -14401.205} C_VEL
LIN {X 0,Y 334.064,Z 263.861,A -85,B 0,C 180,E1 -14402.411,E2 -14402.411} C_VEL
LIN {X 0,Y 333.978,Z 263.877,A -85,B 0,C 180,E1 -14406.039,E2 -14406.039} C_VEL
LIN {X 0,Y 333.908,Z 263.883,A -85,B 0,C 180,E1 -14408.472,E2 -14408.472} C_VEL
LIN {X 0,Y 333.784,Z 263.898,A -85,B 0,C 180,E1 -14412.155,E2 -14412.155} C_VEL
LIN {X 0,Y 333.804,Z 263.9,A -85,B 0,C 180,E1 -14414.634,E2 -14414.634} C_VEL
LIN {X 0,Y 333.749,Z 263.905,A -85,B 0,C 180,E1 -14418.633,E2 -14418.633} C_VEL
LIN {X 0,Y 333.646,Z 263.918,A -85,B 0,C 180,E1 -14422.281,E2 -14422.281} C_VEL
LIN {X 0,Y 333.683,Z 263.917,A -85,B 0,C 180,E1 -14425.089,E2 -14425.089} C_VEL
LIN {X 0,Y 333.623,Z 263.913,A -85,B 0,C 180,E1 -14428.98,E2 -14428.98} C_VEL
LIN {X 0,Y 333.636,Z 263.915,A -85,B 0,C 180,E1 -14432.586,E2 -14432.586} C_VEL
LIN {X 0,Y 333.671,Z 263.921,A -85,B 0,C 180,E1 -14436.14,E2 -14436.14} C_VEL
LIN {X 0,Y 333.598,Z 263.919,A -85,B 0,C 180,E1 -14439.199,E2 -14439.199} C_VEL
LIN {X 0,Y 333.623,Z 263.921,A -85,B 0,C 180,E1 -14442.499,E2 -14442.499} C_VEL
LIN {X 0,Y 333.591,Z 263.927,A -85,B 0,C 180,E1 -14445.955,E2 -14445.955} C_VEL
LIN {X 0,Y 333.599,Z 263.915,A -85,B 0,C 180,E1 -14449.325,E2 -14449.325} C_VEL
LIN {X 0,Y 333.684,Z 264.055,A -85,B 0,C 180,E1 -14453.163,E2 -14453.163} C_VEL
LIN {X 0,Y 336.942,Z 276.273,A -85,B 0,C 180,E1 -14456.221,E2 -14456.221} C_VEL
LIN {X 0,Y 339.466,Z 287.505,A -85,B 0,C 180,E1 -14458.83,E2 -14458.83} C_VEL
LIN {X 0,Y 340.539,Z 293.161,A -85,B 0,C 180,E1 -14460.088,E2 -14460.088} C_VEL
LIN {X 0,Y 339.167,Z 305.739,A -85,B 0,C 180,E1 -14462.545,E2 -14462.545} C_VEL
LIN {X 0,Y 337.934,Z 317.323,A -85,B 0,C 180,E1 -14464.732,E2 -14464.732} C_VEL
LIN {X 0,Y 342.318,Z 345.132,A -85,B 0,C 180,E1 -14465.791,E2 -14465.791} C_VEL
LIN {X 0,Y 345.144,Z 369.381,A -85,B 0,C 180,E1 -14466.575,E2 -14466.575} C_VEL
LIN {X 0,Y 345.284,Z 376.744,A -85,B 0,C 180,E1 -14466.753,E2 -14466.753} C_VEL
LIN {X 0,Y 344.057,Z 428.449,A -85,B 0,C 180,E1 -14467.856,E2 -14467.856} C_VEL
LIN {X 0,Y 343.243,Z 442.036,A -85,B 0,C 180,E1 -14468.373,E2 -14468.373} C_VEL
LIN {X 0,Y 341.925,Z 454.67,A -85,B 0,C 180,E1 -14469.076,E2 -14469.076} C_VEL
LIN {X 0,Y 340.521,Z 465.942,A -85,B 0,C 180,E1 -14469.933,E2 -14469.933} C_VEL
LIN {X 0,Y 338.819,Z 477.633,A -85,B 0,C 180,E1 -14471.089,E2 -14471.089} C_VEL
LIN {X 0,Y 337.202,Z 488.189,A -85,B 0,C 180,E1 -14472.409,E2 -14472.409} C_VEL
LIN {X 0,Y 335.692,Z 497.752,A -85,B 0,C 180,E1 -14473.895,E2 -14473.895} C_VEL
LIN {X 0,Y 334.469,Z 507.031,A -85,B 0,C 180,E1 -14475.706,E2 -14475.706} C_VEL
LIN {X 0,Y 333.397,Z 514.545,A -85,B 0,C 180,E1 -14477.521,E2 -14477.521} C_VEL
LIN {X 0,Y 332.627,Z 521.525,A -85,B 0,C 180,E1 -14479.654,E2 -14479.654} C_VEL
LIN {X 0,Y 332.423,Z 526.197,A -85,B 0,C 180,E1 -14481.489,E2 -14481.489} C_VEL
LIN {X 0,Y 332.485,Z 530.002,A -85,B 0,C 180,E1 -14483.452,E2 -14483.452} C_VEL
LIN {X 0,Y 332.557,Z 532.386,A -85,B 0,C 180,E1 -14485.15,E2 -14485.15} C_VEL
LIN {X 0,Y 332.756,Z 533.577,A -85,B 0,C 180,E1 -14486.367,E2 -14486.367} C_VEL
LIN {X 0,Y 332.864,Z 534.345,A -85,B 0,C 180,E1 -14487.579,E2 -14487.579} C_VEL
LIN {X 0,Y 332.989,Z 534.676,A -85,B 0,C 180,E1 -14489.999,E2 -14489.999} C_VEL
LIN {X 0,Y 332.933,Z 534.186,A -85,B 0,C 180,E1 -14491.209,E2 -14491.209} C_VEL
LIN {X 0,Y 332.922,Z 533.276,A -85,B 0,C 180,E1 -14492.419,E2 -14492.419} C_VEL
LIN {X 0,Y 332.92,Z 531.956,A -85,B 0,C 180,E1 -14493.63,E2 -14493.63} C_VEL
LIN {X 0,Y 332.661,Z 529.093,A -85,B 0,C 180,E1 -14495.455,E2 -14495.455} C_VEL
LIN {X 0,Y 332.559,Z 525.174,A -85,B 0,C 180,E1 -14497.284,E2 -14497.284} C_VEL
LIN {X 0,Y 332.556,Z 520.086,A -85,B 0,C 180,E1 -14499.119,E2 -14499.119} C_VEL
LIN {X 0,Y 332.819,Z 513.698,A -85,B 0,C 180,E1 -14500.955,E2 -14500.955} C_VEL
LIN {X 0,Y 333.375,Z 505.739,A -85,B 0,C 180,E1 -14502.788,E2 -14502.788} C_VEL
LIN {X 0,Y 334.056,Z 497.609,A -85,B 0,C 180,E1 -14504.311,E2 -14504.311} C_VEL
LIN {X 0,Y 335.204,Z 487.749,A -85,B 0,C 180,E1 -14505.816,E2 -14505.816} C_VEL
LIN {X 0,Y 336.306,Z 476.777,A -85,B 0,C 180,E1 -14507.167,E2 -14507.167} C_VEL
LIN {X 0,Y 337.38,Z 466.099,A -85,B 0,C 180,E1 -14508.207,E2 -14508.207} C_VEL
LIN {X 0,Y 338.612,Z 453.276,A -85,B 0,C 180,E1 -14509.158,E2 -14509.158} C_VEL
LIN {X 0,Y 339.535,Z 440.423,A -85,B 0,C 180,E1 -14509.851,E2 -14509.851} C_VEL
LIN {X 0,Y 340.027,Z 427.942,A -85,B 0,C 180,E1 -14510.294,E2 -14510.294} C_VEL
LIN {X 0,Y 340.909,Z 369.899,A -85,B 0,C 180,E1 -14511.523,E2 -14511.523} C_VEL
LIN {X 0,Y 335.872,Z 320.722,A -85,B 0,C 180,E1 -14512.882,E2 -14512.882} C_VEL
LIN {X 0,Y 335.674,Z 318.439,A -85,B 0,C 180,E1 -14513.003,E2 -14513.003} C_VEL
LIN {X 0,Y 337.613,Z 295.874,A -85,B 0,C 180,E1 -14517.255,E2 -14517.255} C_VEL
LIN {X 0,Y 338.338,Z 286.532,A -85,B 0,C 180,E1 -14519.037,E2 -14519.037} C_VEL
LIN {X 0,Y 335.7,Z 272.905,A -85,B 0,C 180,E1 -14521.911,E2 -14521.911} C_VEL
LIN {X 0,Y 333.67,Z 264.008,A -85,B 0,C 180,E1 -14523.927,E2 -14523.927} C_VEL
LIN {X 0,Y 333.637,Z 263.926,A -85,B 0,C 180,E1 -14527.652,E2 -14527.652} C_VEL
LIN {X 0,Y 333.597,Z 263.927,A -85,B 0,C 180,E1 -14530.773,E2 -14530.773} C_VEL
LIN {X 0,Y 333.583,Z 263.925,A -85,B 0,C 180,E1 -14534.249,E2 -14534.249} C_VEL
LIN {X 0,Y 333.628,Z 263.926,A -85,B 0,C 180,E1 -14537.616,E2 -14537.616} C_VEL
LIN {X 0,Y 333.626,Z 263.927,A -85,B 0,C 180,E1 -14541.205,E2 -14541.205} C_VEL
LIN {X 0,Y 333.664,Z 263.92,A -85,B 0,C 180,E1 -14543.86,E2 -14543.86} C_VEL
LIN {X 0,Y 333.628,Z 263.923,A -85,B 0,C 180,E1 -14547.414,E2 -14547.414} C_VEL
LIN {X 0,Y 333.638,Z 263.928,A -85,B 0,C 180,E1 -14551.021,E2 -14551.021} C_VEL
LIN {X 0,Y 333.684,Z 263.92,A -85,B 0,C 180,E1 -14555.087,E2 -14555.087} C_VEL
LIN {X 0,Y 333.645,Z 263.925,A -85,B 0,C 180,E1 -14559.017,E2 -14559.017} C_VEL
LIN {X 0,Y 333.729,Z 263.908,A -85,B 0,C 180,E1 -14561.586,E2 -14561.586} C_VEL
LIN {X 0,Y 333.798,Z 263.903,A -85,B 0,C 180,E1 -14565.577,E2 -14565.577} C_VEL
LIN {X 0,Y 333.804,Z 263.901,A -85,B 0,C 180,E1 -14569.077,E2 -14569.077} C_VEL
LIN {X 0,Y 333.942,Z 263.889,A -85,B 0,C 180,E1 -14572.746,E2 -14572.746} C_VEL
LIN {X 0,Y 333.769,Z 263.907,A -85,B 0,C 180,E1 -14575.169,E2 -14575.169} C_VEL
LIN {X 0,Y 334.057,Z 263.868,A -85,B 0,C 180,E1 -14577.589,E2 -14577.589} C_VEL
LIN {X 0,Y 334.064,Z 263.869,A -85,B 0,C 180,E1 -14581.206,E2 -14581.206} C_VEL
LIN {X 0,Y 334.044,Z 263.876,A -85,B 0,C 180,E1 -14582.412,E2 -14582.412} C_VEL
LIN {X 0,Y 333.941,Z 263.882,A -85,B 0,C 180,E1 -14586.593,E2 -14586.593} C_VEL
LIN {X 0,Y 333.807,Z 263.899,A -85,B 0,C 180,E1 -14589.697,E2 -14589.697} C_VEL
LIN {X 0,Y 333.785,Z 263.904,A -85,B 0,C 180,E1 -14593.392,E2 -14593.392} C_VEL
LIN {X 0,Y 333.708,Z 263.91,A -85,B 0,C 180,E1 -14597.149,E2 -14597.149} C_VEL
LIN {X 0,Y 333.661,Z 263.919,A -85,B 0,C 180,E1 -14599.695,E2 -14599.695} C_VEL
LIN {X 0,Y 333.636,Z 263.924,A -85,B 0,C 180,E1 -14603.593,E2 -14603.593} C_VEL
LIN {X 0,Y 333.62,Z 263.927,A -85,B 0,C 180,E1 -14606.256,E2 -14606.256} C_VEL
LIN {X 0,Y 333.62,Z 263.925,A -85,B 0,C 180,E1 -14608.981,E2 -14608.981} C_VEL
LIN {X 0,Y 333.636,Z 263.921,A -85,B 0,C 180,E1 -14612.588,E2 -14612.588} C_VEL
LIN {X 0,Y 333.666,Z 263.923,A -85,B 0,C 180,E1 -14616.141,E2 -14616.141} C_VEL
LIN {X 0,Y 333.595,Z 263.928,A -85,B 0,C 180,E1 -14619.2,E2 -14619.2} C_VEL
LIN {X 0,Y 333.62,Z 263.915,A -85,B 0,C 180,E1 -14622.5,E2 -14622.5} C_VEL
LIN {X 0,Y 333.588,Z 263.932,A -85,B 0,C 180,E1 -14625.956,E2 -14625.956} C_VEL
LIN {X 0,Y 333.598,Z 263.93,A -85,B 0,C 180,E1 -14629.326,E2 -14629.326} C_VEL
LIN {X 0,Y 333.658,Z 263.914,A -85,B 0,C 180,E1 -14633.17,E2 -14633.17} C_VEL
LIN {X 0,Y 333.67,Z 263.92,A -85,B 0,C 180,E1 -14635.342,E2 -14635.342} C_VEL
LIN {X 0,Y 333.618,Z 263.924,A -85,B 0,C 180,E1 -14638.222,E2 -14638.222} C_VEL
LIN {X 0,Y 333.622,Z 263.923,A -85,B 0,C 180,E1 -14641.021,E2 -14641.021} C_VEL
LIN {X 0,Y 333.657,Z 263.92,A -85,B 0,C 180,E1 -14644.923,E2 -14644.923} C_VEL
LIN {X 0,Y 333.641,Z 263.924,A -85,B 0,C 180,E1 -14649.018,E2 -14649.018} C_VEL
LIN {X 0,Y 333.711,Z 263.905,A -85,B 0,C 180,E1 -14651.586,E2 -14651.586} C_VEL
LIN {X 0,Y 333.737,Z 264.025,A -85,B 0,C 180,E1 -14655.285,E2 -14655.285} C_VEL
LIN {X 0,Y 333.925,Z 264.866,A -85,B 0,C 180,E1 -14655.502,E2 -14655.502} C_VEL
LIN {X 0,Y 339.684,Z 279.127,A -85,B 0,C 180,E1 -14656.216,E2 -14656.216} C_VEL
LIN {X 0,Y 342.184,Z 285.908,A -85,B 0,C 180,E1 -14656.513,E2 -14656.513} C_VEL
LIN {X 0,Y 341.176,Z 351.482,A -85,B 0,C 180,E1 -14657.906,E2 -14657.906} C_VEL
LIN {X 0,Y 340.879,Z 364.894,A -85,B 0,C 180,E1 -14658.442,E2 -14658.442} C_VEL
LIN {X 0,Y 340.436,Z 377.873,A -85,B 0,C 180,E1 -14659.218,E2 -14659.218} C_VEL
LIN {X 0,Y 339.674,Z 389.646,A -85,B 0,C 180,E1 -14660.172,E2 -14660.172} C_VEL
LIN {X 0,Y 338.727,Z 400.929,A -85,B 0,C 180,E1 -14661.349,E2 -14661.349} C_VEL
LIN {X 0,Y 337.887,Z 411.072,A -85,B 0,C 180,E1 -14662.681,E2 -14662.681} C_VEL
LIN {X 0,Y 337.056,Z 419.389,A -85,B 0,C 180,E1 -14664.016,E2 -14664.016} C_VEL
LIN {X 0,Y 336.092,Z 428.407,A -85,B 0,C 180,E1 -14665.803,E2 -14665.803} C_VEL
LIN {X 0,Y 335.176,Z 435.688,A -85,B 0,C 180,E1 -14667.597,E2 -14667.597} C_VEL
LIN {X 0,Y 334.516,Z 441.522,A -85,B 0,C 180,E1 -14669.399,E2 -14669.399} C_VEL
LIN {X 0,Y 334.036,Z 446.134,A -85,B 0,C 180,E1 -14671.206,E2 -14671.206} C_VEL
LIN {X 0,Y 333.587,Z 449.683,A -85,B 0,C 180,E1 -14673.02,E2 -14673.02} C_VEL
LIN {X 0,Y 333.498,Z 452.213,A -85,B 0,C 180,E1 -14674.836,E2 -14674.836} C_VEL
LIN {X 0,Y 333.442,Z 453.419,A -85,B 0,C 180,E1 -14676.05,E2 -14676.05} C_VEL
LIN {X 0,Y 333.415,Z 454.588,A -85,B 0,C 180,E1 -14678.485,E2 -14678.485} C_VEL
LIN {X 0,Y 333.629,Z 454.234,A -85,B 0,C 180,E1 -14680.929,E2 -14680.929} C_VEL
LIN {X 0,Y 333.85,Z 453.429,A -85,B 0,C 180,E1 -14682.153,E2 -14682.153} C_VEL
LIN {X 0,Y 334.136,Z 452.224,A -85,B 0,C 180,E1 -14683.378,E2 -14683.378} C_VEL
LIN {X 0,Y 334.693,Z 449.991,A -85,B 0,C 180,E1 -14684.998,E2 -14684.998} C_VEL
LIN {X 0,Y 335.481,Z 446.006,A -85,B 0,C 180,E1 -14687.055,E2 -14687.055} C_VEL
LIN {X 0,Y 336.404,Z 441.241,A -85,B 0,C 180,E1 -14688.894,E2 -14688.894} C_VEL
LIN {X 0,Y 337.571,Z 435.174,A -85,B 0,C 180,E1 -14690.728,E2 -14690.728} C_VEL
LIN {X 0,Y 338.922,Z 427.559,A -85,B 0,C 180,E1 -14692.558,E2 -14692.558} C_VEL
LIN {X 0,Y 340.212,Z 419.683,A -85,B 0,C 180,E1 -14694.079,E2 -14694.079} C_VEL
LIN {X 0,Y 341.539,Z 410.003,A -85,B 0,C 180,E1 -14695.603,E2 -14695.603} C_VEL
LIN {X 0,Y 342.95,Z 399.16,A -85,B 0,C 180,E1 -14696.962,E2 -14696.962} C_VEL
LIN {X 0,Y 344.047,Z 388.474,A -85,B 0,C 180,E1 -14698.023,E2 -14698.023} C_VEL
LIN {X 0,Y 344.983,Z 376.951,A -85,B 0,C 180,E1 -14698.913,E2 -14698.913} C_VEL
LIN {X 0,Y 345.622,Z 363.765,A -85,B 0,C 180,E1 -14699.67,E2 -14699.67} C_VEL
LIN {X 0,Y 345.918,Z 351.206,A -85,B 0,C 180,E1 -14700.146,E2 -14700.146} C_VEL
LIN {X 0,Y 346.655,Z 309.749,A -85,B 0,C 180,E1 -14701.049,E2 -14701.049} C_VEL
LIN {X 0,Y 347.146,Z 292.082,A -85,B 0,C 180,E1 -14701.412,E2 -14701.412} C_VEL
LIN {X 0,Y 339.726,Z 276.34,A -85,B 0,C 180,E1 -14702.426,E2 -14702.426} C_VEL
LIN {X 0,Y 337.96,Z 274.688,A -85,B 0,C 180,E1 -14702.626,E2 -14702.626} C_VEL
LIN {X 0,Y 331.095,Z 272.723,A -85,B 0,C 180,E1 -14703.319,E2 -14703.319} C_VEL
LIN {X 0,Y 329.79,Z 271.523,A -85,B 0,C 180,E1 -14703.476,E2 -14703.476} C_VEL
LIN {X 0,Y 326.866,Z 265.942,A -85,B 0,C 180,E1 -14703.927,E2 -14703.927} C_VEL
LIN {X 0,Y 326.653,Z 264.913,A -85,B 0,C 180,E1 -14704.176,E2 -14704.176} C_VEL
LIN {X 0,Y 326.623,Z 264.752,A -85,B 0,C 180,E1 -14707.236,E2 -14707.236} C_VEL
LIN {X 0,Y 326.543,Z 264.8,A -85,B 0,C 180,E1 -14711.124,E2 -14711.124} C_VEL
LIN {X 0,Y 326.559,Z 264.807,A -85,B 0,C 180,E1 -14713.526,E2 -14713.526} C_VEL
LIN {X 0,Y 326.57,Z 264.786,A -85,B 0,C 180,E1 -14717.029,E2 -14717.029} C_VEL
LIN {X 0,Y 326.57,Z 264.797,A -85,B 0,C 180,E1 -14720.781,E2 -14720.781} C_VEL
LIN {X 0,Y 326.624,Z 264.774,A -85,B 0,C 180,E1 -14722.952,E2 -14722.952} C_VEL
LIN {X 0,Y 326.605,Z 264.805,A -85,B 0,C 180,E1 -14725.98,E2 -14725.98} C_VEL
LIN {X 0,Y 326.609,Z 264.766,A -85,B 0,C 180,E1 -14729.397,E2 -14729.397} C_VEL
LIN {X 0,Y 326.609,Z 264.802,A -85,B 0,C 180,E1 -14733.135,E2 -14733.135} C_VEL
LIN {X 0,Y 326.627,Z 264.781,A -85,B 0,C 180,E1 -14735.869,E2 -14735.869} C_VEL
LIN {X 0,Y 326.651,Z 264.767,A -85,B 0,C 180,E1 -14739.864,E2 -14739.864} C_VEL
LIN {X 0,Y 326.696,Z 264.791,A -85,B 0,C 180,E1 -14742.472,E2 -14742.472} C_VEL
LIN {X 0,Y 326.755,Z 264.775,A -85,B 0,C 180,E1 -14746.314,E2 -14746.314} C_VEL
LIN {X 0,Y 326.778,Z 264.767,A -85,B 0,C 180,E1 -14750.092,E2 -14750.092} C_VEL
LIN {X 0,Y 326.934,Z 264.761,A -85,B 0,C 180,E1 -14753.829,E2 -14753.829} C_VEL
LIN {X 0,Y 327.001,Z 264.745,A -85,B 0,C 180,E1 -14757.536,E2 -14757.536} C_VEL
LIN {X 0,Y 327.023,Z 264.739,A -85,B 0,C 180,E1 -14761.231,E2 -14761.231} C_VEL
LIN {X 0,Y 326.753,Z 264.78,A -85,B 0,C 180,E1 -14763.699,E2 -14763.699} C_VEL
LIN {X 0,Y 326.933,Z 264.753,A -85,B 0,C 180,E1 -14766.17,E2 -14766.17} C_VEL
LIN {X 0,Y 326.778,Z 264.78,A -85,B 0,C 180,E1 -14769.907,E2 -14769.907} C_VEL
LIN {X 0,Y 326.752,Z 264.773,A -85,B 0,C 180,E1 -14773.686,E2 -14773.686} C_VEL
LIN {X 0,Y 326.659,Z 264.788,A -85,B 0,C 180,E1 -14777.53,E2 -14777.53} C_VEL
LIN {X 0,Y 326.642,Z 264.796,A -85,B 0,C 180,E1 -14780.136,E2 -14780.136} C_VEL
LIN {X 0,Y 326.624,Z 264.799,A -85,B 0,C 180,E1 -14784.131,E2 -14784.131} C_VEL
LIN {X 0,Y 326.591,Z 264.78,A -85,B 0,C 180,E1 -14788.081,E2 -14788.081} C_VEL
LIN {X 0,Y 326.563,Z 264.809,A -85,B 0,C 180,E1 -14791.098,E2 -14791.098} C_VEL
LIN {X 0,Y 326.602,Z 264.782,A -85,B 0,C 180,E1 -14794.02,E2 -14794.02} C_VEL
LIN {X 0,Y 326.619,Z 264.797,A -85,B 0,C 180,E1 -14797.237,E2 -14797.237} C_VEL
LIN {X 0,Y 326.54,Z 264.814,A -85,B 0,C 180,E1 -14801.124,E2 -14801.124} C_VEL
LIN {X 0,Y 326.556,Z 264.799,A -85,B 0,C 180,E1 -14803.527,E2 -14803.527} C_VEL
LIN {X 0,Y 326.569,Z 264.8,A -85,B 0,C 180,E1 -14807.029,E2 -14807.029} C_VEL
LIN {X 0,Y 326.569,Z 264.778,A -85,B 0,C 180,E1 -14810.782,E2 -14810.782} C_VEL
LIN {X 0,Y 326.642,Z 265.003,A -85,B 0,C 180,E1 -14812.603,E2 -14812.603} C_VEL
LIN {X 0,Y 330.055,Z 277.61,A -85,B 0,C 180,E1 -14815.841,E2 -14815.841} C_VEL
LIN {X 0,Y 332.878,Z 290.295,A -85,B 0,C 180,E1 -14818.851,E2 -14818.851} C_VEL
LIN {X 0,Y 333.731,Z 295.305,A -85,B 0,C 180,E1 -14819.983,E2 -14819.983} C_VEL
LIN {X 0,Y 332.014,Z 309.275,A -85,B 0,C 180,E1 -14822.754,E2 -14822.754} C_VEL
LIN {X 0,Y 331.255,Z 316.394,A -85,B 0,C 180,E1 -14824.108,E2 -14824.108} C_VEL
LIN {X 0,Y 335.392,Z 342.089,A -85,B 0,C 180,E1 -14825.128,E2 -14825.128} C_VEL
LIN {X 0,Y 338.367,Z 365.883,A -85,B 0,C 180,E1 -14825.942,E2 -14825.942} C_VEL
LIN {X 0,Y 338.971,Z 374.806,A -85,B 0,C 180,E1 -14826.2,E2 -14826.2} C_VEL
LIN {X 0,Y 337.583,Z 428.09,A -85,B 0,C 180,E1 -14827.358,E2 -14827.358} C_VEL
LIN {X 0,Y 336.751,Z 441.704,A -85,B 0,C 180,E1 -14827.895,E2 -14827.895} C_VEL
LIN {X 0,Y 335.307,Z 454.706,A -85,B 0,C 180,E1 -14828.643,E2 -14828.643} C_VEL
LIN {X 0,Y 333.854,Z 465.743,A -85,B 0,C 180,E1 -14829.514,E2 -14829.514} C_VEL
LIN {X 0,Y 332.105,Z 477.311,A -85,B 0,C 180,E1 -14830.691,E2 -14830.691} C_VEL
LIN {X 0,Y 330.393,Z 487.771,A -85,B 0,C 180,E1 -14832.035,E2 -14832.035} C_VEL
LIN {X 0,Y 328.819,Z 497.235,A -85,B 0,C 180,E1 -14833.549,E2 -14833.549} C_VEL
LIN {X 0,Y 327.538,Z 506.446,A -85,B 0,C 180,E1 -14835.397,E2 -14835.397} C_VEL
LIN {X 0,Y 326.415,Z 513.909,A -85,B 0,C 180,E1 -14837.25,E2 -14837.25} C_VEL
LIN {X 0,Y 325.575,Z 520.824,A -85,B 0,C 180,E1 -14839.427,E2 -14839.427} C_VEL
LIN {X 0,Y 325.344,Z 525.459,A -85,B 0,C 180,E1 -14841.303,E2 -14841.303} C_VEL
LIN {X 0,Y 325.408,Z 529.457,A -85,B 0,C 180,E1 -14843.457,E2 -14843.457} C_VEL
LIN {X 0,Y 325.477,Z 531.594,A -85,B 0,C 180,E1 -14845.045,E2 -14845.045} C_VEL
LIN {X 0,Y 325.686,Z 532.762,A -85,B 0,C 180,E1 -14846.288,E2 -14846.288} C_VEL
LIN {X 0,Y 325.814,Z 533.518,A -85,B 0,C 180,E1 -14847.527,E2 -14847.527} C_VEL
LIN {X 0,Y 325.94,Z 533.814,A -85,B 0,C 180,E1 -14849.999,E2 -14849.999} C_VEL
LIN {X 0,Y 325.882,Z 533.296,A -85,B 0,C 180,E1 -14851.235,E2 -14851.235} C_VEL
LIN {X 0,Y 325.875,Z 532.371,A -85,B 0,C 180,E1 -14852.472,E2 -14852.472} C_VEL
LIN {X 0,Y 325.842,Z 531.03,A -85,B 0,C 180,E1 -14853.709,E2 -14853.709} C_VEL
LIN {X 0,Y 325.593,Z 528.132,A -85,B 0,C 180,E1 -14855.573,E2 -14855.573} C_VEL
LIN {X 0,Y 325.472,Z 524.17,A -85,B 0,C 180,E1 -14857.443,E2 -14857.443} C_VEL
LIN {X 0,Y 325.534,Z 518.083,A -85,B 0,C 180,E1 -14859.631,E2 -14859.631} C_VEL
LIN {X 0,Y 325.921,Z 511.38,A -85,B 0,C 180,E1 -14861.505,E2 -14861.505} C_VEL
LIN {X 0,Y 326.558,Z 503.054,A -85,B 0,C 180,E1 -14863.376,E2 -14863.376} C_VEL
LIN {X 0,Y 327.495,Z 493.838,A -85,B 0,C 180,E1 -14865.051,E2 -14865.051} C_VEL
LIN {X 0,Y 328.431,Z 484.174,A -85,B 0,C 180,E1 -14866.47,E2 -14866.47} C_VEL
LIN {X 0,Y 329.66,Z 473.921,A -85,B 0,C 180,E1 -14867.685,E2 -14867.685} C_VEL
LIN {X 0,Y 330.822,Z 462.733,A -85,B 0,C 180,E1 -14868.742,E2 -14868.742} C_VEL
LIN {X 0,Y 331.941,Z 450.327,A -85,B 0,C 180,E1 -14869.639,E2 -14869.639} C_VEL
LIN {X 0,Y 332.892,Z 437.203,A -85,B 0,C 180,E1 -14870.305,E2 -14870.305} C_VEL
LIN {X 0,Y 333.348,Z 424.578,A -85,B 0,C 180,E1 -14870.719,E2 -14870.719} C_VEL
LIN {X 0,Y 334.123,Z 370.19,A -85,B 0,C 180,E1 -14871.887,E2 -14871.887} C_VEL
LIN {X 0,Y 329.209,Z 321.871,A -85,B 0,C 180,E1 -14873.256,E2 -14873.256} C_VEL
LIN {X 0,Y 328.74,Z 317.598,A -85,B 0,C 180,E1 -14873.439,E2 -14873.439} C_VEL
LIN {X 0,Y 330.708,Z 296.322,A -85,B 0,C 180,E1 -14877.529,E2 -14877.529} C_VEL
LIN {X 0,Y 331.425,Z 287.787,A -85,B 0,C 180,E1 -14879.19,E2 -14879.19} C_VEL
LIN {X 0,Y 328.824,Z 274.584,A -85,B 0,C 180,E1 -14882.04,E2 -14882.04} C_VEL
LIN {X 0,Y 326.635,Z 264.895,A -85,B 0,C 180,E1 -14884.271,E2 -14884.271} C_VEL
LIN {X 0,Y 326.616,Z 264.802,A -85,B 0,C 180,E1 -14887.236,E2 -14887.236} C_VEL
LIN {X 0,Y 326.537,Z 264.809,A -85,B 0,C 180,E1 -14891.123,E2 -14891.123} C_VEL
LIN {X 0,Y 326.552,Z 264.804,A -85,B 0,C 180,E1 -14893.525,E2 -14893.525} C_VEL
LIN {X 0,Y 326.564,Z 264.803,A -85,B 0,C 180,E1 -14897.028,E2 -14897.028} C_VEL
LIN {X 0,Y 326.573,Z 264.804,A -85,B 0,C 180,E1 -14901.384,E2 -14901.384} C_VEL
LIN {X 0,Y 326.609,Z 264.802,A -85,B 0,C 180,E1 -14904.851,E2 -14904.851} C_VEL
LIN {X 0,Y 326.593,Z 264.798,A -85,B 0,C 180,E1 -14907.454,E2 -14907.454} C_VEL
LIN {X 0,Y 326.578,Z 264.802,A -85,B 0,C 180,E1 -14910.333,E2 -14910.333} C_VEL
LIN {X 0,Y 326.623,Z 264.796,A -85,B 0,C 180,E1 -14914.511,E2 -14914.511} C_VEL
LIN {X 0,Y 326.6,Z 264.802,A -85,B 0,C 180,E1 -14918.542,E2 -14918.542} C_VEL
LIN {X 0,Y 326.652,Z 264.791,A -85,B 0,C 180,E1 -14922.47,E2 -14922.47} C_VEL
LIN {X 0,Y 326.746,Z 264.783,A -85,B 0,C 180,E1 -14926.314,E2 -14926.314} C_VEL
LIN {X 0,Y 326.771,Z 264.775,A -85,B 0,C 180,E1 -14930.093,E2 -14930.093} C_VEL
LIN {X 0,Y 326.926,Z 264.759,A -85,B 0,C 180,E1 -14933.83,E2 -14933.83} C_VEL
LIN {X 0,Y 327,Z 264.747,A -85,B 0,C 180,E1 -14937.537,E2 -14937.537} C_VEL
LIN {X 0,Y 327.032,Z 264.744,A -85,B 0,C 180,E1 -14941.232,E2 -14941.232} C_VEL
LIN {X 0,Y 326.722,Z 264.784,A -85,B 0,C 180,E1 -14943.7,E2 -14943.7} C_VEL
LIN {X 0,Y 326.902,Z 264.76,A -85,B 0,C 180,E1 -14946.585,E2 -14946.585} C_VEL
LIN {X 0,Y 326.77,Z 264.776,A -85,B 0,C 180,E1 -14949.908,E2 -14949.908} C_VEL
LIN {X 0,Y 326.748,Z 264.781,A -85,B 0,C 180,E1 -14953.686,E2 -14953.686} C_VEL
LIN {X 0,Y 326.653,Z 264.788,A -85,B 0,C 180,E1 -14957.531,E2 -14957.531} C_VEL
LIN {X 0,Y 326.605,Z 264.799,A -85,B 0,C 180,E1 -14961.458,E2 -14961.458} C_VEL
LIN {X 0,Y 326.592,Z 264.798,A -85,B 0,C 180,E1 -14965.492,E2 -14965.492} C_VEL
LIN {X 0,Y 326.581,Z 264.805,A -85,B 0,C 180,E1 -14968.258,E2 -14968.258} C_VEL
LIN {X 0,Y 326.565,Z 264.803,A -85,B 0,C 180,E1 -14971.099,E2 -14971.099} C_VEL
LIN {X 0,Y 326.599,Z 264.801,A -85,B 0,C 180,E1 -14974.021,E2 -14974.021} C_VEL
LIN {X 0,Y 326.615,Z 264.798,A -85,B 0,C 180,E1 -14977.238,E2 -14977.238} C_VEL
LIN {X 0,Y 326.537,Z 264.802,A -85,B 0,C 180,E1 -14981.125,E2 -14981.125} C_VEL
LIN {X 0,Y 326.553,Z 264.796,A -85,B 0,C 180,E1 -14983.528,E2 -14983.528} C_VEL
LIN {X 0,Y 326.567,Z 264.803,A -85,B 0,C 180,E1 -14987.031,E2 -14987.031} C_VEL
LIN {X 0,Y 326.568,Z 264.801,A -85,B 0,C 180,E1 -14990.783,E2 -14990.783} C_VEL
LIN {X 0,Y 326.608,Z 264.796,A -85,B 0,C 180,E1 -14994.481,E2 -14994.481} C_VEL
LIN {X 0,Y 326.602,Z 264.804,A -85,B 0,C 180,E1 -14997.456,E2 -14997.456} C_VEL
LIN {X 0,Y 326.574,Z 264.799,A -85,B 0,C 180,E1 -15000.334,E2 -15000.334} C_VEL
LIN {X 0,Y 326.594,Z 264.803,A -85,B 0,C 180,E1 -15003.136,E2 -15003.136} C_VEL
LIN {X 0,Y 326.593,Z 264.805,A -85,B 0,C 180,E1 -15007.212,E2 -15007.212} C_VEL
LIN {X 0,Y 326.631,Z 264.781,A -85,B 0,C 180,E1 -15011.216,E2 -15011.216} C_VEL
LIN {X 0,Y 326.71,Z 264.956,A -85,B 0,C 180,E1 -15014.882,E2 -15014.882} C_VEL
LIN {X 0,Y 326.875,Z 265.785,A -85,B 0,C 180,E1 -15015.071,E2 -15015.071} C_VEL
LIN {X 0,Y 333.359,Z 281.711,A -85,B 0,C 180,E1 -15015.883,E2 -15015.883} C_VEL
LIN {X 0,Y 335.392,Z 287.266,A -85,B 0,C 180,E1 -15016.133,E2 -15016.133} C_VEL
LIN {X 0,Y 334.45,Z 352.473,A -85,B 0,C 180,E1 -15017.554,E2 -15017.554} C_VEL
LIN {X 0,Y 334.132,Z 365.633,A -85,B 0,C 180,E1 -15018.09,E2 -15018.09} C_VEL
LIN {X 0,Y 333.708,Z 378.085,A -85,B 0,C 180,E1 -15018.844,E2 -15018.844} C_VEL
LIN {X 0,Y 332.904,Z 390.047,A -85,B 0,C 180,E1 -15019.817,E2 -15019.817} C_VEL
LIN {X 0,Y 331.919,Z 401.412,A -85,B 0,C 180,E1 -15021.017,E2 -15021.017} C_VEL
LIN {X 0,Y 331.045,Z 411.615,A -85,B 0,C 180,E1 -15022.376,E2 -15022.376} C_VEL
LIN {X 0,Y 330.072,Z 420.835,A -85,B 0,C 180,E1 -15023.889,E2 -15023.889} C_VEL
LIN {X 0,Y 329.087,Z 429.727,A -85,B 0,C 180,E1 -15025.714,E2 -15025.714} C_VEL
LIN {X 0,Y 328.154,Z 436.925,A -85,B 0,C 180,E1 -15027.546,E2 -15027.546} C_VEL
LIN {X 0,Y 327.477,Z 442.686,A -85,B 0,C 180,E1 -15029.386,E2 -15029.386} C_VEL
LIN {X 0,Y 326.996,Z 447.23,A -85,B 0,C 180,E1 -15031.232,E2 -15031.232} C_VEL
LIN {X 0,Y 326.633,Z 449.663,A -85,B 0,C 180,E1 -15032.467,E2 -15032.467} C_VEL
LIN {X 0,Y 326.444,Z 451.638,A -85,B 0,C 180,E1 -15033.704,E2 -15033.704} C_VEL
LIN {X 0,Y 326.461,Z 453.189,A -85,B 0,C 180,E1 -15034.94,E2 -15034.94} C_VEL
LIN {X 0,Y 326.402,Z 454.352,A -85,B 0,C 180,E1 -15036.181,E2 -15036.181} C_VEL
LIN {X 0,Y 326.375,Z 455.457,A -85,B 0,C 180,E1 -15038.67,E2 -15038.67} C_VEL
LIN {X 0,Y 326.482,Z 455.441,A -85,B 0,C 180,E1 -15039.917,E2 -15039.917} C_VEL
LIN {X 0,Y 326.632,Z 455.028,A -85,B 0,C 180,E1 -15041.166,E2 -15041.166} C_VEL
LIN {X 0,Y 327.2,Z 452.949,A -85,B 0,C 180,E1 -15043.667,E2 -15043.667} C_VEL
LIN {X 0,Y 327.743,Z 450.844,A -85,B 0,C 180,E1 -15045.21,E2 -15045.21} C_VEL
LIN {X 0,Y 328.618,Z 446.611,A -85,B 0,C 180,E1 -15047.422,E2 -15047.422} C_VEL
LIN {X 0,Y 329.616,Z 441.776,A -85,B 0,C 180,E1 -15049.298,E2 -15049.298} C_VEL
LIN {X 0,Y 330.865,Z 435.634,A -85,B 0,C 180,E1 -15051.168,E2 -15051.168} C_VEL
LIN {X 0,Y 332.281,Z 427.888,A -85,B 0,C 180,E1 -15053.035,E2 -15053.035} C_VEL
LIN {X 0,Y 333.678,Z 419.904,A -85,B 0,C 180,E1 -15054.581,E2 -15054.581} C_VEL
LIN {X 0,Y 335.051,Z 410.098,A -85,B 0,C 180,E1 -15056.135,E2 -15056.135} C_VEL
LIN {X 0,Y 336.373,Z 400.402,A -85,B 0,C 180,E1 -15057.365,E2 -15057.365} C_VEL
LIN {X 0,Y 337.524,Z 389.854,A -85,B 0,C 180,E1 -15058.444,E2 -15058.444} C_VEL
LIN {X 0,Y 338.513,Z 378.431,A -85,B 0,C 180,E1 -15059.353,E2 -15059.353} C_VEL
LIN {X 0,Y 339.197,Z 365.02,A -85,B 0,C 180,E1 -15060.147,E2 -15060.147} C_VEL
LIN {X 0,Y 339.546,Z 352.155,A -85,B 0,C 180,E1 -15060.648,E2 -15060.648} C_VEL
LIN {X 0,Y 340.334,Z 309.702,A -85,B 0,C 180,E1 -15061.588,E2 -15061.588} C_VEL
LIN {X 0,Y 340.765,Z 293.943,A -85,B 0,C 180,E1 -15061.919,E2 -15061.919} C_VEL
LIN {X 0,Y 332.693,Z 277.113,A -85,B 0,C 180,E1 -15063.058,E2 -15063.058} C_VEL
LIN {X 0,Y 329.79,Z 271.523,A -85,B 0,C 180,E1 -15063.476,E2 -15063.476} C_VEL
LIN {X 0,Y 327.456,Z 268.904,A -85,B 0,C 180,E1 -15063.846,E2 -15063.846} C_VEL
LIN {X 0,Y 324.935,Z 267.232,A -85,B 0,C 180,E1 -15064.347,E2 -15064.347} C_VEL
LIN {X 0,Y 321.893,Z 266.061,A -85,B 0,C 180,E1 -15065.159,E2 -15065.159} C_VEL
LIN {X 0,Y 319.873,Z 265.661,A -85,B 0,C 180,E1 -15066.097,E2 -15066.097} C_VEL
LIN {X 0,Y 319.546,Z 265.629,A -85,B 0,C 180,E1 -15066.597,E2 -15066.597} C_VEL
LIN {X 0,Y 319.529,Z 265.686,A -85,B 0,C 180,E1 -15069.661,E2 -15069.661} C_VEL
LIN {X 0,Y 319.519,Z 265.682,A -85,B 0,C 180,E1 -15073.459,E2 -15073.459} C_VEL
LIN {X 0,Y 319.549,Z 265.66,A -85,B 0,C 180,E1 -15077.015,E2 -15077.015} C_VEL
LIN {X 0,Y 319.513,Z 265.68,A -85,B 0,C 180,E1 -15080.365,E2 -15080.365} C_VEL
LIN {X 0,Y 319.578,Z 265.668,A -85,B 0,C 180,E1 -15084.457,E2 -15084.457} C_VEL
LIN {X 0,Y 319.522,Z 265.661,A -85,B 0,C 180,E1 -15088.137,E2 -15088.137} C_VEL
LIN {X 0,Y 319.567,Z 265.665,A -85,B 0,C 180,E1 -15091.604,E2 -15091.604} C_VEL
LIN {X 0,Y 319.57,Z 265.67,A -85,B 0,C 180,E1 -15095.301,E2 -15095.301} C_VEL
LIN {X 0,Y 319.562,Z 265.633,A -85,B 0,C 180,E1 -15098.045,E2 -15098.045} C_VEL
LIN {X 0,Y 319.686,Z 265.652,A -85,B 0,C 180,E1 -15100.962,E2 -15100.962} C_VEL
LIN {X 0,Y 319.728,Z 265.646,A -85,B 0,C 180,E1 -15105.276,E2 -15105.276} C_VEL
LIN {X 0,Y 319.71,Z 265.658,A -85,B 0,C 180,E1 -15108.589,E2 -15108.589} C_VEL
LIN {X 0,Y 319.847,Z 265.642,A -85,B 0,C 180,E1 -15112.424,E2 -15112.424} C_VEL
LIN {X 0,Y 319.708,Z 265.656,A -85,B 0,C 180,E1 -15114.955,E2 -15114.955} C_VEL
LIN {X 0,Y 320.007,Z 265.622,A -85,B 0,C 180,E1 -15118.741,E2 -15118.741} C_VEL
LIN {X 0,Y 319.953,Z 265.619,A -85,B 0,C 180,E1 -15122.518,E2 -15122.518} C_VEL
LIN {X 0,Y 319.89,Z 265.63,A -85,B 0,C 180,E1 -15126.306,E2 -15126.306} C_VEL
LIN {X 0,Y 319.73,Z 265.657,A -85,B 0,C 180,E1 -15130.128,E2 -15130.128} C_VEL
LIN {X 0,Y 319.726,Z 265.65,A -85,B 0,C 180,E1 -15133.992,E2 -15133.992} C_VEL
LIN {X 0,Y 319.62,Z 265.664,A -85,B 0,C 180,E1 -15137.929,E2 -15137.929} C_VEL
LIN {X 0,Y 319.59,Z 265.675,A -85,B 0,C 180,E1 -15140.6,E2 -15140.6} C_VEL
LIN {X 0,Y 319.545,Z 265.681,A -85,B 0,C 180,E1 -15143.321,E2 -15143.321} C_VEL
LIN {X 0,Y 319.562,Z 265.666,A -85,B 0,C 180,E1 -15146.094,E2 -15146.094} C_VEL
LIN {X 0,Y 319.519,Z 265.669,A -85,B 0,C 180,E1 -15148.94,E2 -15148.94} C_VEL
LIN {X 0,Y 319.516,Z 265.681,A -85,B 0,C 180,E1 -15151.863,E2 -15151.863} C_VEL
LIN {X 0,Y 319.576,Z 265.674,A -85,B 0,C 180,E1 -15155.543,E2 -15155.543} C_VEL
LIN {X 0,Y 319.525,Z 265.674,A -85,B 0,C 180,E1 -15159.662,E2 -15159.662} C_VEL
LIN {X 0,Y 319.515,Z 265.675,A -85,B 0,C 180,E1 -15163.46,E2 -15163.46} C_VEL
LIN {X 0,Y 319.548,Z 265.674,A -85,B 0,C 180,E1 -15167.016,E2 -15167.016} C_VEL
LIN {X 0,Y 319.532,Z 265.658,A -85,B 0,C 180,E1 -15171.586,E2 -15171.586} C_VEL
LIN {X 0,Y 319.565,Z 265.919,A -85,B 0,C 180,E1 -15171.991,E2 -15171.991} C_VEL
LIN {X 0,Y 322.464,Z 276.266,A -85,B 0,C 180,E1 -15174.757,E2 -15174.757} C_VEL
LIN {X 0,Y 325.314,Z 288.447,A -85,B 0,C 180,E1 -15177.774,E2 -15177.774} C_VEL
LIN {X 0,Y 326.905,Z 296.372,A -85,B 0,C 180,E1 -15179.64,E2 -15179.64} C_VEL
LIN {X 0,Y 325.602,Z 307.399,A -85,B 0,C 180,E1 -15181.886,E2 -15181.886} C_VEL
LIN {X 0,Y 324.626,Z 315.527,A -85,B 0,C 180,E1 -15183.464,E2 -15183.464} C_VEL
LIN {X 0,Y 328.692,Z 340.733,A -85,B 0,C 180,E1 -15184.495,E2 -15184.495} C_VEL
LIN {X 0,Y 331.742,Z 364.258,A -85,B 0,C 180,E1 -15185.336,E2 -15185.336} C_VEL
LIN {X 0,Y 332.6,Z 374.5,A -85,B 0,C 180,E1 -15185.655,E2 -15185.655} C_VEL
LIN {X 0,Y 331.228,Z 426.631,A -85,B 0,C 180,E1 -15186.805,E2 -15186.805} C_VEL
LIN {X 0,Y 330.389,Z 439.863,A -85,B 0,C 180,E1 -15187.322,E2 -15187.322} C_VEL
LIN {X 0,Y 329.047,Z 452.605,A -85,B 0,C 180,E1 -15188.051,E2 -15188.051} C_VEL
LIN {X 0,Y 327.496,Z 463.966,A -85,B 0,C 180,E1 -15188.933,E2 -15188.933} C_VEL
LIN {X 0,Y 325.587,Z 475.701,A -85,B 0,C 180,E1 -15190.125,E2 -15190.125} C_VEL
LIN {X 0,Y 323.851,Z 486.287,A -85,B 0,C 180,E1 -15191.495,E2 -15191.495} C_VEL
LIN {X 0,Y 322.252,Z 494.973,A -85,B 0,C 180,E1 -15192.877,E2 -15192.877} C_VEL
LIN {X 0,Y 320.946,Z 503.186,A -85,B 0,C 180,E1 -15194.473,E2 -15194.473} C_VEL
LIN {X 0,Y 319.96,Z 509.762,A -85,B 0,C 180,E1 -15196.018,E2 -15196.018} C_VEL
LIN {X 0,Y 319.02,Z 516.439,A -85,B 0,C 180,E1 -15197.919,E2 -15197.919} C_VEL
LIN {X 0,Y 318.413,Z 521.802,A -85,B 0,C 180,E1 -15199.829,E2 -15199.829} C_VEL
LIN {X 0,Y 318.235,Z 526.027,A -85,B 0,C 180,E1 -15201.746,E2 -15201.746} C_VEL
LIN {X 0,Y 318.363,Z 529.216,A -85,B 0,C 180,E1 -15203.663,E2 -15203.663} C_VEL
LIN {X 0,Y 318.401,Z 530.797,A -85,B 0,C 180,E1 -15204.934,E2 -15204.934} C_VEL
LIN {X 0,Y 318.616,Z 531.948,A -85,B 0,C 180,E1 -15206.205,E2 -15206.205} C_VEL
LIN {X 0,Y 318.764,Z 532.691,A -85,B 0,C 180,E1 -15207.472,E2 -15207.472} C_VEL
LIN {X 0,Y 318.777,Z 533.02,A -85,B 0,C 180,E1 -15208.736,E2 -15208.736} C_VEL
LIN {X 0,Y 318.891,Z 532.947,A -85,B 0,C 180,E1 -15209.999,E2 -15209.999} C_VEL
LIN {X 0,Y 318.832,Z 532.406,A -85,B 0,C 180,E1 -15211.263,E2 -15211.263} C_VEL
LIN {X 0,Y 318.828,Z 531.465,A -85,B 0,C 180,E1 -15212.526,E2 -15212.526} C_VEL
LIN {X 0,Y 318.767,Z 530.102,A -85,B 0,C 180,E1 -15213.792,E2 -15213.792} C_VEL
LIN {X 0,Y 318.529,Z 527.169,A -85,B 0,C 180,E1 -15215.697,E2 -15215.697} C_VEL
LIN {X 0,Y 318.398,Z 523.166,A -85,B 0,C 180,E1 -15217.61,E2 -15217.61} C_VEL
LIN {X 0,Y 318.472,Z 517.013,A -85,B 0,C 180,E1 -15219.847,E2 -15219.847} C_VEL
LIN {X 0,Y 318.879,Z 510.259,A -85,B 0,C 180,E1 -15221.762,E2 -15221.762} C_VEL
LIN {X 0,Y 319.62,Z 501.888,A -85,B 0,C 180,E1 -15223.672,E2 -15223.672} C_VEL
LIN {X 0,Y 320.488,Z 493.344,A -85,B 0,C 180,E1 -15225.256,E2 -15225.256} C_VEL
LIN {X 0,Y 321.438,Z 484.007,A -85,B 0,C 180,E1 -15226.676,E2 -15226.676} C_VEL
LIN {X 0,Y 322.693,Z 473.906,A -85,B 0,C 180,E1 -15227.916,E2 -15227.916} C_VEL
LIN {X 0,Y 323.883,Z 462.918,A -85,B 0,C 180,E1 -15228.994,E2 -15228.994} C_VEL
LIN {X 0,Y 325.028,Z 450.803,A -85,B 0,C 180,E1 -15229.91,E2 -15229.91} C_VEL
LIN {X 0,Y 326.057,Z 437.567,A -85,B 0,C 180,E1 -15230.626,E2 -15230.626} C_VEL
LIN {X 0,Y 326.583,Z 424.207,A -85,B 0,C 180,E1 -15231.086,E2 -15231.086} C_VEL
LIN {X 0,Y 327.407,Z 370.89,A -85,B 0,C 180,E1 -15232.254,E2 -15232.254} C_VEL
LIN {X 0,Y 322.663,Z 323.58,A -85,B 0,C 180,E1 -15233.626,E2 -15233.626} C_VEL
LIN {X 0,Y 321.854,Z 317.049,A -85,B 0,C 180,E1 -15233.858,E2 -15233.858} C_VEL
LIN {X 0,Y 323.795,Z 296.763,A -85,B 0,C 180,E1 -15237.816,E2 -15237.816} C_VEL
LIN {X 0,Y 324.458,Z 288.89,A -85,B 0,C 180,E1 -15239.385,E2 -15239.385} C_VEL
LIN {X 0,Y 321.776,Z 275.482,A -85,B 0,C 180,E1 -15242.349,E2 -15242.349} C_VEL
LIN {X 0,Y 319.618,Z 265.763,A -85,B 0,C 180,E1 -15244.647,E2 -15244.647} C_VEL
LIN {X 0,Y 319.517,Z 265.682,A -85,B 0,C 180,E1 -15248.014,E2 -15248.014} C_VEL
LIN {X 0,Y 319.497,Z 265.688,A -85,B 0,C 180,E1 -15251.591,E2 -15251.591} C_VEL
LIN {X 0,Y 319.478,Z 265.68,A -85,B 0,C 180,E1 -15254.743,E2 -15254.743} C_VEL
LIN {X 0,Y 319.543,Z 265.677,A -85,B 0,C 180,E1 -15257.015,E2 -15257.015} C_VEL
LIN {X 0,Y 319.538,Z 265.679,A -85,B 0,C 180,E1 -15260.37,E2 -15260.37} C_VEL
LIN {X 0,Y 319.569,Z 265.676,A -85,B 0,C 180,E1 -15264.457,E2 -15264.457} C_VEL
LIN {X 0,Y 319.509,Z 265.678,A -85,B 0,C 180,E1 -15268.136,E2 -15268.136} C_VEL
LIN {X 0,Y 319.557,Z 265.677,A -85,B 0,C 180,E1 -15271.605,E2 -15271.605} C_VEL
LIN {X 0,Y 319.561,Z 265.676,A -85,B 0,C 180,E1 -15275.301,E2 -15275.301} C_VEL
LIN {X 0,Y 319.554,Z 265.677,A -85,B 0,C 180,E1 -15278.045,E2 -15278.045} C_VEL
LIN {X 0,Y 319.603,Z 265.666,A -85,B 0,C 180,E1 -15282.07,E2 -15282.07} C_VEL
LIN {X 0,Y 319.72,Z 265.657,A -85,B 0,C 180,E1 -15286.007,E2 -15286.007} C_VEL
LIN {X 0,Y 319.723,Z 265.651,A -85,B 0,C 180,E1 -15289.872,E2 -15289.872} C_VEL
LIN {X 0,Y 319.884,Z 265.636,A -85,B 0,C 180,E1 -15293.693,E2 -15293.693} C_VEL
LIN {X 0,Y 319.947,Z 265.625,A -85,B 0,C 180,E1 -15297.482,E2 -15297.482} C_VEL
LIN {X 0,Y 320,Z 265.62,A -85,B 0,C 180,E1 -15301.259,E2 -15301.259} C_VEL
LIN {X 0,Y 319.885,Z 265.639,A -85,B 0,C 180,E1 -15306.307,E2 -15306.307} C_VEL
LIN {X 0,Y 319.723,Z 265.654,A -85,B 0,C 180,E1 -15310.129,E2 -15310.129} C_VEL
LIN {X 0,Y 319.722,Z 265.659,A -85,B 0,C 180,E1 -15313.993,E2 -15313.993} C_VEL
LIN {X 0,Y 319.604,Z 265.667,A -85,B 0,C 180,E1 -15317.93,E2 -15317.93} C_VEL
LIN {X 0,Y 319.556,Z 265.68,A -85,B 0,C 180,E1 -15321.956,E2 -15321.956} C_VEL
LIN {X 0,Y 319.541,Z 265.678,A -85,B 0,C 180,E1 -15326.097,E2 -15326.097} C_VEL
LIN {X 0,Y 319.516,Z 265.682,A -85,B 0,C 180,E1 -15328.941,E2 -15328.941} C_VEL
LIN {X 0,Y 319.516,Z 265.686,A -85,B 0,C 180,E1 -15331.864,E2 -15331.864} C_VEL
LIN {X 0,Y 319.571,Z 265.676,A -85,B 0,C 180,E1 -15335.543,E2 -15335.543} C_VEL
LIN {X 0,Y 319.523,Z 265.683,A -85,B 0,C 180,E1 -15339.663,E2 -15339.663} C_VEL
LIN {X 0,Y 319.513,Z 265.669,A -85,B 0,C 180,E1 -15343.461,E2 -15343.461} C_VEL
LIN {X 0,Y 319.546,Z 265.677,A -85,B 0,C 180,E1 -15347.017,E2 -15347.017} C_VEL
LIN {X 0,Y 319.511,Z 265.68,A -85,B 0,C 180,E1 -15350.367,E2 -15350.367} C_VEL
LIN {X 0,Y 319.575,Z 265.672,A -85,B 0,C 180,E1 -15354.459,E2 -15354.459} C_VEL
LIN {X 0,Y 319.518,Z 265.68,A -85,B 0,C 180,E1 -15358.138,E2 -15358.138} C_VEL
LIN {X 0,Y 319.541,Z 265.682,A -85,B 0,C 180,E1 -15361.615,E2 -15361.615} C_VEL
LIN {X 0,Y 319.54,Z 265.678,A -85,B 0,C 180,E1 -15365.3,E2 -15365.3} C_VEL
LIN {X 0,Y 319.561,Z 265.676,A -85,B 0,C 180,E1 -15368.046,E2 -15368.046} C_VEL
LIN {X 0,Y 319.581,Z 265.661,A -85,B 0,C 180,E1 -15372.07,E2 -15372.07} C_VEL
LIN {X 0,Y 319.666,Z 265.894,A -85,B 0,C 180,E1 -15374.45,E2 -15374.45} C_VEL
LIN {X 0,Y 319.946,Z 267.064,A -85,B 0,C 180,E1 -15374.643,E2 -15374.643} C_VEL
LIN {X 0,Y 326.872,Z 283.834,A -85,B 0,C 180,E1 -15375.516,E2 -15375.516} C_VEL
LIN {X 0,Y 328.795,Z 289.074,A -85,B 0,C 180,E1 -15375.76,E2 -15375.76} C_VEL
LIN {X 0,Y 327.73,Z 352.947,A -85,B 0,C 180,E1 -15377.171,E2 -15377.171} C_VEL
LIN {X 0,Y 327.395,Z 366.343,A -85,B 0,C 180,E1 -15377.723,E2 -15377.723} C_VEL
LIN {X 0,Y 326.915,Z 379.383,A -85,B 0,C 180,E1 -15378.531,E2 -15378.531} C_VEL
LIN {X 0,Y 326.149,Z 390.429,A -85,B 0,C 180,E1 -15379.447,E2 -15379.447} C_VEL
LIN {X 0,Y 325.125,Z 401.88,A -85,B 0,C 180,E1 -15380.671,E2 -15380.671} C_VEL
LIN {X 0,Y 324.21,Z 412.15,A -85,B 0,C 180,E1 -15382.057,E2 -15382.057} C_VEL
LIN {X 0,Y 323.299,Z 420.571,A -85,B 0,C 180,E1 -15383.447,E2 -15383.447} C_VEL
LIN {X 0,Y 322.388,Z 428.343,A -85,B 0,C 180,E1 -15384.998,E2 -15384.998} C_VEL
LIN {X 0,Y 321.385,Z 435.966,A -85,B 0,C 180,E1 -15386.867,E2 -15386.867} C_VEL
LIN {X 0,Y 320.62,Z 442.07,A -85,B 0,C 180,E1 -15388.745,E2 -15388.745} C_VEL
LIN {X 0,Y 320.072,Z 446.924,A -85,B 0,C 180,E1 -15390.63,E2 -15390.63} C_VEL
LIN {X 0,Y 319.568,Z 450.7,A -85,B 0,C 180,E1 -15392.521,E2 -15392.521} C_VEL
LIN {X 0,Y 319.395,Z 452.643,A -85,B 0,C 180,E1 -15393.785,E2 -15393.785} C_VEL
LIN {X 0,Y 319.425,Z 454.165,A -85,B 0,C 180,E1 -15395.049,E2 -15395.049} C_VEL
LIN {X 0,Y 319.344,Z 455.276,A -85,B 0,C 180,E1 -15396.318,E2 -15396.318} C_VEL
LIN {X 0,Y 319.337,Z 456.325,A -85,B 0,C 180,E1 -15398.862,E2 -15398.862} C_VEL
LIN {X 0,Y 319.456,Z 456.282,A -85,B 0,C 180,E1 -15400.137,E2 -15400.137} C_VEL
LIN {X 0,Y 319.647,Z 455.812,A -85,B 0,C 180,E1 -15401.413,E2 -15401.413} C_VEL
LIN {X 0,Y 320.276,Z 453.676,A -85,B 0,C 180,E1 -15403.968,E2 -15403.968} C_VEL
LIN {X 0,Y 320.786,Z 451.715,A -85,B 0,C 180,E1 -15405.422,E2 -15405.422} C_VEL
LIN {X 0,Y 321.795,Z 447.217,A -85,B 0,C 180,E1 -15407.804,E2 -15407.804} C_VEL
LIN {X 0,Y 322.843,Z 442.316,A -85,B 0,C 180,E1 -15409.72,E2 -15409.72} C_VEL
LIN {X 0,Y 324.188,Z 436.092,A -85,B 0,C 180,E1 -15411.626,E2 -15411.626} C_VEL
LIN {X 0,Y 325.678,Z 428.22,A -85,B 0,C 180,E1 -15413.53,E2 -15413.53} C_VEL
LIN {X 0,Y 327.15,Z 420.131,A -85,B 0,C 180,E1 -15415.105,E2 -15415.105} C_VEL
LIN {X 0,Y 328.623,Z 410.198,A -85,B 0,C 180,E1 -15416.686,E2 -15416.686} C_VEL
LIN {X 0,Y 329.979,Z 400.309,A -85,B 0,C 180,E1 -15417.941,E2 -15417.941} C_VEL
LIN {X 0,Y 331.216,Z 389.455,A -85,B 0,C 180,E1 -15419.037,E2 -15419.037} C_VEL
LIN {X 0,Y 332.113,Z 379.201,A -85,B 0,C 180,E1 -15419.859,E2 -15419.859} C_VEL
LIN {X 0,Y 332.792,Z 366.343,A -85,B 0,C 180,E1 -15420.639,E2 -15420.639} C_VEL
LIN {X 0,Y 333.192,Z 353.53,A -85,B 0,C 180,E1 -15421.158,E2 -15421.158} C_VEL
LIN {X 0,Y 333.971,Z 312.794,A -85,B 0,C 180,E1 -15422.082,E2 -15422.082} C_VEL
LIN {X 0,Y 334.432,Z 295.914,A -85,B 0,C 180,E1 -15422.443,E2 -15422.443} C_VEL
LIN {X 0,Y 327.226,Z 280.938,A -85,B 0,C 180,E1 -15423.496,E2 -15423.496} C_VEL
LIN {X 0,Y 319.764,Z 266.541,A -85,B 0,C 180,E1 -15424.661,E2 -15424.661} C_VEL
LIN {X 0,Y 319.593,Z 265.726,A -85,B 0,C 180,E1 -15424.955,E2 -15424.955} C_VEL
LIN {X 0,Y 319.546,Z 265.629,A -85,B 0,C 180,E1 -15426.597,E2 -15426.597} C_VEL
LIN {X 0,Y 318.841,Z 265.73,A -85,B 0,C 180,E1 -15427.649,E2 -15427.649} C_VEL
LIN {X 0,Y 315.957,Z 266.123,A -85,B 0,C 180,E1 -15429.361,E2 -15429.361} C_VEL
LIN {X 0,Y 313.545,Z 266.423,A -85,B 0,C 180,E1 -15430.749,E2 -15430.749} C_VEL
LIN {X 0,Y 312.529,Z 266.541,A -85,B 0,C 180,E1 -15431.824,E2 -15431.824} C_VEL
LIN {X 0,Y 312.456,Z 266.549,A -85,B 0,C 180,E1 -15432.188,E2 -15432.188} C_VEL
LIN {X 0,Y 312.456,Z 266.547,A -85,B 0,C 180,E1 -15436.035,E2 -15436.035} C_VEL
LIN {X 0,Y 312.454,Z 266.566,A -85,B 0,C 180,E1 -15439.885,E2 -15439.885} C_VEL
LIN {X 0,Y 312.533,Z 266.54,A -85,B 0,C 180,E1 -15444.05,E2 -15444.05} C_VEL
LIN {X 0,Y 312.5,Z 266.55,A -85,B 0,C 180,E1 -15447.333,E2 -15447.333} C_VEL
LIN {X 0,Y 312.497,Z 266.538,A -85,B 0,C 180,E1 -15451.294,E2 -15451.294} C_VEL
LIN {X 0,Y 312.544,Z 266.55,A -85,B 0,C 180,E1 -15454.707,E2 -15454.707} C_VEL
LIN {X 0,Y 312.531,Z 266.511,A -85,B 0,C 180,E1 -15458.912,E2 -15458.912} C_VEL
LIN {X 0,Y 312.635,Z 266.535,A -85,B 0,C 180,E1 -15461.656,E2 -15461.656} C_VEL
LIN {X 0,Y 312.69,Z 266.522,A -85,B 0,C 180,E1 -15465.686,E2 -15465.686} C_VEL
LIN {X 0,Y 312.681,Z 266.527,A -85,B 0,C 180,E1 -15469.641,E2 -15469.641} C_VEL
LIN {X 0,Y 312.79,Z 266.519,A -85,B 0,C 180,E1 -15472.252,E2 -15472.252} C_VEL
LIN {X 0,Y 312.679,Z 266.531,A -85,B 0,C 180,E1 -15474.841,E2 -15474.841} C_VEL
LIN {X 0,Y 312.974,Z 266.498,A -85,B 0,C 180,E1 -15478.713,E2 -15478.713} C_VEL
LIN {X 0,Y 312.902,Z 266.497,A -85,B 0,C 180,E1 -15482.574,E2 -15482.574} C_VEL
LIN {X 0,Y 312.832,Z 266.509,A -85,B 0,C 180,E1 -15486.449,E2 -15486.449} C_VEL
LIN {X 0,Y 312.746,Z 266.521,A -85,B 0,C 180,E1 -15489.05,E2 -15489.05} C_VEL
LIN {X 0,Y 312.627,Z 266.529,A -85,B 0,C 180,E1 -15492.991,E2 -15492.991} C_VEL
LIN {X 0,Y 312.617,Z 266.545,A -85,B 0,C 180,E1 -15495.651,E2 -15495.651} C_VEL
LIN {X 0,Y 312.559,Z 266.553,A -85,B 0,C 180,E1 -15499.711,E2 -15499.711} C_VEL
LIN {X 0,Y 312.516,Z 266.551,A -85,B 0,C 180,E1 -15502.778,E2 -15502.778} C_VEL
LIN {X 0,Y 312.523,Z 266.545,A -85,B 0,C 180,E1 -15505.907,E2 -15505.907} C_VEL
LIN {X 0,Y 312.463,Z 266.558,A -85,B 0,C 180,E1 -15509.658,E2 -15509.658} C_VEL
LIN {X 0,Y 312.516,Z 266.536,A -85,B 0,C 180,E1 -15513.689,E2 -15513.689} C_VEL
LIN {X 0,Y 312.507,Z 266.554,A -85,B 0,C 180,E1 -15517.388,E2 -15517.388} C_VEL
LIN {X 0,Y 312.437,Z 266.568,A -85,B 0,C 180,E1 -15520.717,E2 -15520.717} C_VEL
LIN {X 0,Y 312.447,Z 266.562,A -85,B 0,C 180,E1 -15524.21,E2 -15524.21} C_VEL
LIN {X 0,Y 312.452,Z 266.567,A -85,B 0,C 180,E1 -15527.925,E2 -15527.925} C_VEL
LIN {X 0,Y 312.503,Z 266.712,A -85,B 0,C 180,E1 -15531.302,E2 -15531.302} C_VEL
LIN {X 0,Y 315.909,Z 278.906,A -85,B 0,C 180,E1 -15534.661,E2 -15534.661} C_VEL
LIN {X 0,Y 318.527,Z 290.158,A -85,B 0,C 180,E1 -15537.515,E2 -15537.515} C_VEL
LIN {X 0,Y 320.016,Z 297.466,A -85,B 0,C 180,E1 -15539.281,E2 -15539.281} C_VEL
LIN {X 0,Y 319.433,Z 304.112,A -85,B 0,C 180,E1 -15540.69,E2 -15540.69} C_VEL
LIN {X 0,Y 318.048,Z 314.433,A -85,B 0,C 180,E1 -15542.774,E2 -15542.774} C_VEL
LIN {X 0,Y 322.3,Z 340.844,A -85,B 0,C 180,E1 -15543.898,E2 -15543.898} C_VEL
LIN {X 0,Y 325.464,Z 365.368,A -85,B 0,C 180,E1 -15544.801,E2 -15544.801} C_VEL
LIN {X 0,Y 326.239,Z 375.802,A -85,B 0,C 180,E1 -15545.126,E2 -15545.126} C_VEL
LIN {X 0,Y 324.808,Z 426.597,A -85,B 0,C 180,E1 -15546.277,E2 -15546.277} C_VEL
LIN {X 0,Y 323.873,Z 440.314,A -85,B 0,C 180,E1 -15546.839,E2 -15546.839} C_VEL
LIN {X 0,Y 322.482,Z 452.694,A -85,B 0,C 180,E1 -15547.58,E2 -15547.58} C_VEL
LIN {X 0,Y 320.861,Z 463.794,A -85,B 0,C 180,E1 -15548.476,E2 -15548.476} C_VEL
LIN {X 0,Y 318.902,Z 475.395,A -85,B 0,C 180,E1 -15549.69,E2 -15549.69} C_VEL
LIN {X 0,Y 317.083,Z 485.883,A -85,B 0,C 180,E1 -15551.085,E2 -15551.085} C_VEL
LIN {X 0,Y 315.443,Z 494.493,A -85,B 0,C 180,E1 -15552.496,E2 -15552.496} C_VEL
LIN {X 0,Y 313.837,Z 503.901,A -85,B 0,C 180,E1 -15554.411,E2 -15554.411} C_VEL
LIN {X 0,Y 312.799,Z 510.361,A -85,B 0,C 180,E1 -15556.023,E2 -15556.023} C_VEL
LIN {X 0,Y 311.721,Z 517.662,A -85,B 0,C 180,E1 -15558.292,E2 -15558.292} C_VEL
LIN {X 0,Y 311.253,Z 522.592,A -85,B 0,C 180,E1 -15560.25,E2 -15560.25} C_VEL
LIN {X 0,Y 311.171,Z 526.43,A -85,B 0,C 180,E1 -15562.211,E2 -15562.211} C_VEL
LIN {X 0,Y 311.268,Z 528.447,A -85,B 0,C 180,E1 -15563.517,E2 -15563.517} C_VEL
LIN {X 0,Y 311.327,Z 529.998,A -85,B 0,C 180,E1 -15564.819,E2 -15564.819} C_VEL
LIN {X 0,Y 311.549,Z 531.135,A -85,B 0,C 180,E1 -15566.119,E2 -15566.119} C_VEL
LIN {X 0,Y 311.713,Z 531.865,A -85,B 0,C 180,E1 -15567.415,E2 -15567.415} C_VEL
LIN {X 0,Y 311.724,Z 532.178,A -85,B 0,C 180,E1 -15568.708,E2 -15568.708} C_VEL
LIN {X 0,Y 311.843,Z 532.075,A -85,B 0,C 180,E1 -15569.999,E2 -15569.999} C_VEL
LIN {X 0,Y 311.782,Z 531.515,A -85,B 0,C 180,E1 -15571.291,E2 -15571.291} C_VEL
LIN {X 0,Y 311.78,Z 530.557,A -85,B 0,C 180,E1 -15572.583,E2 -15572.583} C_VEL
LIN {X 0,Y 311.693,Z 529.174,A -85,B 0,C 180,E1 -15573.878,E2 -15573.878} C_VEL
LIN {X 0,Y 311.462,Z 526.204,A -85,B 0,C 180,E1 -15575.827,E2 -15575.827} C_VEL
LIN {X 0,Y 311.326,Z 522.159,A -85,B 0,C 180,E1 -15577.784,E2 -15577.784} C_VEL
LIN {X 0,Y 311.426,Z 515.941,A -85,B 0,C 180,E1 -15580.072,E2 -15580.072} C_VEL
LIN {X 0,Y 311.868,Z 509.139,A -85,B 0,C 180,E1 -15582.031,E2 -15582.031} C_VEL
LIN {X 0,Y 312.679,Z 500.717,A -85,B 0,C 180,E1 -15583.982,E2 -15583.982} C_VEL
LIN {X 0,Y 313.569,Z 492.098,A -85,B 0,C 180,E1 -15585.601,E2 -15585.601} C_VEL
LIN {X 0,Y 314.78,Z 481.47,A -85,B 0,C 180,E1 -15587.206,E2 -15587.206} C_VEL
LIN {X 0,Y 316.027,Z 470.984,A -85,B 0,C 180,E1 -15588.475,E2 -15588.475} C_VEL
LIN {X 0,Y 317.416,Z 459.535,A -85,B 0,C 180,E1 -15589.565,E2 -15589.565} C_VEL
LIN {X 0,Y 318.471,Z 447.76,A -85,B 0,C 180,E1 -15590.422,E2 -15590.422} C_VEL
LIN {X 0,Y 319.395,Z 434.19,A -85,B 0,C 180,E1 -15591.119,E2 -15591.119} C_VEL
LIN {X 0,Y 319.931,Z 420.694,A -85,B 0,C 180,E1 -15591.546,E2 -15591.546} C_VEL
LIN {X 0,Y 320.646,Z 371.036,A -85,B 0,C 180,E1 -15592.653,E2 -15592.653} C_VEL
LIN {X 0,Y 315.857,Z 323.397,A -85,B 0,C 180,E1 -15594.074,E2 -15594.074} C_VEL
LIN {X 0,Y 315.03,Z 316.027,A -85,B 0,C 180,E1 -15594.351,E2 -15594.351} C_VEL
LIN {X 0,Y 316.894,Z 297.202,A -85,B 0,C 180,E1 -15598.116,E2 -15598.116} C_VEL
LIN {X 0,Y 317.517,Z 290.715,A -85,B 0,C 180,E1 -15599.433,E2 -15599.433} C_VEL
LIN {X 0,Y 315.282,Z 278.818,A -85,B 0,C 180,E1 -15602.106,E2 -15602.106} C_VEL
LIN {X 0,Y 312.564,Z 266.647,A -85,B 0,C 180,E1 -15605.033,E2 -15605.033} C_VEL
LIN {X 0,Y 312.45,Z 266.557,A -85,B 0,C 180,E1 -15609.034,E2 -15609.034} C_VEL
LIN {X 0,Y 312.458,Z 266.562,A -85,B 0,C 180,E1 -15612.435,E2 -15612.435} C_VEL
LIN {X 0,Y 312.449,Z 266.556,A -85,B 0,C 180,E1 -15616.035,E2 -15616.035} C_VEL
LIN {X 0,Y 312.447,Z 266.563,A -85,B 0,C 180,E1 -15619.885,E2 -15619.885} C_VEL
LIN {X 0,Y 312.525,Z 266.553,A -85,B 0,C 180,E1 -15624.05,E2 -15624.05} C_VEL
LIN {X 0,Y 312.49,Z 266.554,A -85,B 0,C 180,E1 -15627.332,E2 -15627.332} C_VEL
LIN {X 0,Y 312.488,Z 266.56,A -85,B 0,C 180,E1 -15631.294,E2 -15631.294} C_VEL
LIN {X 0,Y 312.536,Z 266.551,A -85,B 0,C 180,E1 -15634.707,E2 -15634.707} C_VEL
LIN {X 0,Y 312.509,Z 266.559,A -85,B 0,C 180,E1 -15638.911,E2 -15638.911} C_VEL
LIN {X 0,Y 312.567,Z 266.548,A -85,B 0,C 180,E1 -15643.004,E2 -15643.004} C_VEL
LIN {X 0,Y 312.674,Z 266.534,A -85,B 0,C 180,E1 -15645.686,E2 -15645.686} C_VEL
LIN {X 0,Y 312.674,Z 266.529,A -85,B 0,C 180,E1 -15649.641,E2 -15649.641} C_VEL
LIN {X 0,Y 312.783,Z 266.519,A -85,B 0,C 180,E1 -15652.252,E2 -15652.252} C_VEL
LIN {X 0,Y 312.677,Z 266.537,A -85,B 0,C 180,E1 -15654.842,E2 -15654.842} C_VEL
LIN {X 0,Y 312.955,Z 266.495,A -85,B 0,C 180,E1 -15658.713,E2 -15658.713} C_VEL
LIN {X 0,Y 312.967,Z 266.496,A -85,B 0,C 180,E1 -15661.287,E2 -15661.287} C_VEL
LIN {X 0,Y 312.818,Z 266.516,A -85,B 0,C 180,E1 -15666.549,E2 -15666.549} C_VEL
LIN {X 0,Y 312.673,Z 266.534,A -85,B 0,C 180,E1 -15670.359,E2 -15670.359} C_VEL
LIN {X 0,Y 312.658,Z 266.535,A -85,B 0,C 180,E1 -15674.865,E2 -15674.865} C_VEL
LIN {X 0,Y 312.539,Z 266.548,A -85,B 0,C 180,E1 -15679.194,E2 -15679.194} C_VEL
LIN {X 0,Y 312.509,Z 266.555,A -85,B 0,C 180,E1 -15682.777,E2 -15682.777} C_VEL
LIN {X 0,Y 312.474,Z 266.556,A -85,B 0,C 180,E1 -15686.733,E2 -15686.733} C_VEL
LIN {X 0,Y 312.461,Z 266.563,A -85,B 0,C 180,E1 -15689.659,E2 -15689.659} C_VEL
LIN {X 0,Y 312.513,Z 266.553,A -85,B 0,C 180,E1 -15693.69,E2 -15693.69} C_VEL
LIN {X 0,Y 312.503,Z 266.557,A -85,B 0,C 180,E1 -15697.389,E2 -15697.389} C_VEL
LIN {X 0,Y 312.435,Z 266.557,A -85,B 0,C 180,E1 -15700.719,E2 -15700.719} C_VEL
LIN {X 0,Y 312.445,Z 266.554,A -85,B 0,C 180,E1 -15704.212,E2 -15704.212} C_VEL
LIN {X 0,Y 312.45,Z 266.566,A -85,B 0,C 180,E1 -15707.926,E2 -15707.926} C_VEL
LIN {X 0,Y 312.472,Z 266.549,A -85,B 0,C 180,E1 -15711.926,E2 -15711.926} C_VEL
LIN {X 0,Y 312.527,Z 266.55,A -85,B 0,C 180,E1 -15714.221,E2 -15714.221} C_VEL
LIN {X 0,Y 312.498,Z 266.56,A -85,B 0,C 180,E1 -15717.335,E2 -15717.335} C_VEL
LIN {X 0,Y 312.481,Z 266.557,A -85,B 0,C 180,E1 -15721.301,E2 -15721.301} C_VEL
LIN {X 0,Y 312.521,Z 266.551,A -85,B 0,C 180,E1 -15724.707,E2 -15724.707} C_VEL
LIN {X 0,Y 312.54,Z 266.555,A -85,B 0,C 180,E1 -15727.527,E2 -15727.527} C_VEL
LIN {X 0,Y 312.544,Z 266.53,A -85,B 0,C 180,E1 -15731.652,E2 -15731.652} C_VEL
LIN {X 0,Y 312.585,Z 266.718,A -85,B 0,C 180,E1 -15733.942,E2 -15733.942} C_VEL
LIN {X 0,Y 312.85,Z 267.804,A -85,B 0,C 180,E1 -15734.157,E2 -15734.157} C_VEL
LIN {X 0,Y 320.64,Z 286.557,A -85,B 0,C 180,E1 -15735.164,E2 -15735.164} C_VEL
LIN {X 0,Y 322.091,Z 290.512,A -85,B 0,C 180,E1 -15735.354,E2 -15735.354} C_VEL
LIN {X 0,Y 321.025,Z 352.752,A -85,B 0,C 180,E1 -15736.754,E2 -15736.754} C_VEL
LIN {X 0,Y 320.751,Z 365.188,A -85,B 0,C 180,E1 -15737.244,E2 -15737.244} C_VEL
LIN {X 0,Y 320.281,Z 378.454,A -85,B 0,C 180,E1 -15738.049,E2 -15738.049} C_VEL
LIN {X 0,Y 319.407,Z 390.795,A -85,B 0,C 180,E1 -15739.061,E2 -15739.061} C_VEL
LIN {X 0,Y 318.345,Z 402.346,A -85,B 0,C 180,E1 -15740.31,E2 -15740.31} C_VEL
LIN {X 0,Y 317.377,Z 412.683,A -85,B 0,C 180,E1 -15741.725,E2 -15741.725} C_VEL
LIN {X 0,Y 316.32,Z 422.032,A -85,B 0,C 180,E1 -15743.302,E2 -15743.302} C_VEL
LIN {X 0,Y 315.237,Z 431.026,A -85,B 0,C 180,E1 -15745.205,E2 -15745.205} C_VEL
